EC00432=798156,1112951
EC00433=798156,1112951
EC00434=798156,1112951
EC00435=798156,1112951
EC00436=798156,1112951
EC00437=798156,1112951
EC00438=798156,1112951
EC00439=798156,1112951
EC00440=798156,1112951
EC00441=798156,1112951
EC00442=798156,1112951
EC00443=798156,1112951
EC00444=798156,1112951
EC00445=798156,1112951
EC00446=798156,1112951
EC00447=798156,1112951
EC00448=798156,1112951
EC00449=798156,1112951
EC00450=798156,1112951
EC00451=798156,1112951
EC00452=798156,1112951
EC00453=798156,1112951
EC00454=798156,1112951
EC00455=798156,1112951
EC00456=798156,1112951
EC00457=798156,1112951
EC00458=798156,1112951
EC00459=798156,1112951
EC00460=798156,1112951
EC00461=798156,1112951
EC00462=798156,1112951
EC00463=798156,1112951
EC00464=798156,1112951
EC00465=798156,1112951
EC00466=798156,1112951
EC00467=798156,1112951
EC00468=798156,1112951
EC00469=798156,1112951
EC00470=798156,1112951
EC00471=798156,1112951
EC00472=798155,1112950
EC00473=798155,1112950
EC00474=798156,1112951
EC00475=798156,1112951
EC00476=798156,1112951
EC00477=798156,1112951
EC00478=798156,1112951
EC00479=798156,1112951
EC00480=798155,1112951
EC00481=798155,1112951
EC00482=798156,1112951
EC00483=798156,1112951
EC00484=798156,1112951
EC00485=798156,1112951
EC00486=798156,1112951
EC00487=798156,1112951
EC00488=798156,1112951
EC00489=798156,1112951
EC00490=798155,1112950
EC00491=798156,1112951
EC00492=798156,1112951
EC00493=798156,1112951
EC00494=798156,1112951
EC00495=798156,1112951
EC00496=798156,1112951
EC00497=798156,1112951
EC00498=798156,1112951
EC00499=798156,1112951
EC00500=798156,1112951
EC00501=798156,1112951
EC00502=798156,1112951
EC00503=798156,1112951
EC00504=798156,1112951
EC00505=798156,1112951
EC00506=798156,1112951
EC00507=798155,1112950
EC00508=798156,1112951
EC00509=798156,1112951
EC00510=798156,1112951
EC00511=798156,1112951
EC00512=798156,1112951
EC00513=798156,1112951
EC00514=798156,1112951
EC00515=798156,1112951
EC00516=798156,1112951
EC00517=798156,1112951
EC00518=798155,1112950
EC00519=798156,1112951
EC00520=798156,1112951
EC00521=798156,1112951
EC00522=798156,1112951
EC00523=798156,1112951
EC00524=798156,1112951
EC00525=798156,1112951
EC00526=798156,1112951
EC00527=798156,1112951
EC00528=798156,1112951
EC00529=798156,1112951
EC00530=798156,1112951
EC00531=798156,1112951
EC00532=798156,1112951
EC00533=798156,1112951
EC00534=798156,1112951
EC00535=798156,1112951
EC00536=798156,1112951
EC00537=798156,1112951
EC00538=798156,1112951
EC00539=798156,1112951
EC00540=798156,1112951
EC00541=798156,1112951
EC00542=798156,1112951
EC00543=798156,1112951
EC00544=798156,1112951
EC00545=798156,1112951
EC00546=798156,1112951
EC00547=798156,1112951
EC00548=798156,1112951
EC00549=798156,1112951
EC00550=798156,1112951
EC00551=798155,1112950
EC00552=798156,1112951
EC00553=798156,1112951
EC00554=798154,1112949
EC00555=798156,1112951
EC00556=798156,1112951
EC00557=798156,1112951
EC00558=798156,1112951
EC00559=798156,1112951
EC00560=798156,1112951
EC00561=798156,1112951
EC00562=798156,1112951
EC00563=798156,1112951
EC00564=798156,1112951
EC00565=798156,1112951
EC00566=798156,1112951
EC00567=798156,1112951
EC00568=798156,1112951
EC00569=798156,1112951
EC00570=798156,1112951
EC00571=798156,1112951
EC00572=798156,1112951
EC00573=798156,1112951
EC00574=798156,1112951
EC00575=798156,1112951
EC00576=798156,1112951
EC00577=798156,1112951
EC00578=798156,1112951
EC00579=798156,1112951
EC00580=798156,1112951
EC00581=798156,1112951
EC00582=798156,1112951
EC00583=798156,1112951
EC00584=798156,1112951
EC00585=798156,1112951
EC00586=798156,1112951
EC00587=798156,1112951
EC00588=798156,1112951
EC00589=798156,1112951
EC00590=798156,1112951
EC00591=798156,1112951
EC00592=798156,1112951
EC00593=798156,1112951
EC00594=798156,1112951
EC00595=798156,1112951
EC00596=798156,1112951
EC00597=798156,1112951
EC00598=798156,1112951
EC00599=798156,1112951
EC00600=798156,1112951
EC00601=798156,1112951
EC00602=798156,1112951
EC00603=798156,1112951
EC00604=798156,1112951
EC00605=798156,1112951
EC00606=798156,1112951
EC00607=798156,1112951
EC00608=798156,1112951
EC00609=798156,1112951
EC00610=798156,1112951
EC00611=798156,1112951
EC00612=798156,1112951
EC00613=798156,1112951
EC00614=798156,1112951
EC00615=798156,1112951
EC00616=798156,1112951
EC00617=798156,1112951
EC00618=798156,1112951
EC00619=798155,1112951
EC00620=798156,1112951
EC00621=798156,1112951
EC00622=798156,1112951
EC00623=798156,1112951
EC00624=798156,1112951
EC00625=798156,1112951
EC00626=798156,1112951
EC00627=798156,1112951
EC00628=798156,1112951
EC00629=798156,1112951
EC00630=798156,1112951
EC00631=798156,1112951
EC00632=798156,1112951
EC00633=798156,1112951
EC00634=798156,1112951
EC00635=798156,1112951
EC00636=798156,1112951
EC00637=798156,1112951
EC00638=798156,1112951
EC00639=798156,1112951
EC00640=798156,1112951
EC00641=798156,1112951
EC00642=798156,1112951
EC00643=798156,1112951
EC00644=798156,1112951
EC00645=798156,1112951
EC00646=798156,1112951
EC00647=798156,1112951
EC00648=798156,1112951
EC00649=798156,1112951
EC00650=798156,1112951
EC00651=798156,1112951
EC00652=798156,1112951
EC00653=798156,1112951
EC00654=798156,1112951
EC00655=798156,1112951
EC00656=798156,1112951
EC00657=798156,1112951
EC00658=798156,1112951
EC00659=798156,1112951
EC00660=798156,1112951
EC00661=798156,1112951
EC00662=798156,1112951
EC00663=798156,1112951
EC00664=798156,1112951
EC00665=798156,1112951
EC00666=798156,1112951
EC00667=798156,1112951
EC00668=798156,1112951
EC00669=798156,1112951
EC00670=798156,1112951
EC00671=798156,1112951
EC00672=798156,1112951
EC00673=798156,1112951
EC00674=798156,1112951
EC00675=798156,1112951
EC00676=798156,1112951
EC00677=798156,1112951
EC00678=798156,1112951
EC00679=798156,1112951
EC00680=798156,1112951
EC00681=798156,1112951
EC00682=798156,1112951
EC00683=798156,1112951
EC00684=798156,1112951
EC00685=798156,1112951
EC00686=798156,1112951
EC00687=798156,1112951
EC00688=798156,1112951
EC00689=798156,1112951
EC00690=798156,1112951
EC00691=798156,1112951
EC00692=798156,1112951
EC00693=798156,1112951
EC00694=798156,1112951
EC00695=798156,1112951
EC00696=798156,1112951
EC00697=798156,1112951
EC00698=798156,1112951
EC00699=798156,1112951
EC00700=798156,1112951
EC00701=798156,1112951
EC00702=798156,1112951
EC00703=798156,1112951
EC00704=798156,1112951
EC00705=798156,1112951
EC00706=798156,1112951
EC00707=798155,1112950
EC00708=798155,1112950
EC00709=798155,1112950
EC00710=798156,1112951
EC00711=798156,1112951
EC00712=798156,1112951
EC00713=798156,1112951
EC00714=798156,1112951
EC00715=798156,1112951
EC00716=798156,1112951
EC00717=798156,1112951
EC00718=798156,1112951
EC00719=798156,1112951
EC00720=798156,1112951
EC00721=798156,1112951
EC00722=798156,1112951
EC00723=798156,1112951
EC00724=798156,1112951
EC00725=798156,1112951
EC00726=798156,1112951
EC00727=798156,1112951
EC00728=798156,1112951
EC00729=798156,1112951
EC00730=798156,1112951
EC00731=798156,1112951
EC00732=798156,1112951
EC00733=798156,1112951
EC00734=798156,1112951
EC00735=798156,1112951
EC00736=798156,1112951
EC00737=798156,1112951
EC00738=798156,1112951
EC00739=798156,1112951
EC00740=798156,1112951
EC00741=798156,1112951
EC00742=798156,1112951
EC00743=798156,1112951
EC00744=798156,1112951
EC00745=798156,1112951
EC00746=798156,1112951
EC00747=798156,1112951
EC00748=798156,1112951
EC00749=798156,1112951
EC00750=798156,1112951
EC00751=798156,1112951
EC00752=798156,1112951
EC00753=798156,1112951
EC00754=798155,1112950
EC00755=798156,1112951
EC00756=798156,1112951
EC00757=798156,1112951
EC00758=798156,1112951
EC00759=798156,1112951
EC00760=798156,1112951
EC00761=798156,1112951
EC00762=798156,1112951
EC00763=798156,1112951
EC00764=798156,1112951
EC00765=798156,1112951
EC00766=798156,1112951
EC00767=798156,1112951
EC00768=798156,1112951
EC00769=798156,1112951
EC00770=798156,1112951
EC00771=798156,1112951
EC00772=798156,1112951
EC00773=798156,1112951
EC00774=798156,1112951
EC00775=798156,1112951
EC00776=798156,1112951
EC00777=798156,1112951
EC00778=798156,1112951
EC00779=798156,1112951
EC00780=798156,1112951
EC00781=798156,1112951
EC00782=798156,1112951
EC00783=798156,1112951
EC00784=798156,1112951
EC00785=798156,1112951
EC00786=798156,1112951
EC00787=798156,1112951
EC00788=798156,1112951
EC00789=798156,1112951
EC00790=798156,1112951
EC00791=798156,1112951
EC00792=798156,1112951
EC00793=798156,1112951
EC00794=798156,1112951
EC00795=798156,1112951
EC00796=798156,1112951
EC00797=798156,1112951
EC00798=798156,1112951
EC00799=798156,1112951
EC00800=798156,1112951
EC00801=798156,1112951
EC00802=798156,1112951
EC00803=798156,1112951
EC00804=798156,1112951
EC00805=798156,1112951
EC00806=798156,1112951
EC00807=798156,1112951
EC00808=798156,1112951
EC00809=798156,1112951
EC00810=798156,1112951
EC00811=798156,1112951
EC00812=798156,1112951
EC00813=798156,1112951
EC00814=798156,1112951
EC00815=798156,1112951
EC00816=798156,1112951
EC00817=798156,1112951
EC00818=798156,1112951
EC00819=798156,1112951
EC00820=798156,1112951
EC00821=798156,1112951
EC00822=798156,1112951
EC00823=798156,1112951
EC00824=798156,1112951
EC00825=798156,1112951
EC00826=798156,1112951
EC00827=798156,1112951
EC00828=798156,1112951
EC00829=798156,1112951
EC00830=798156,1112951
EC00831=798156,1112951
EC00832=798156,1112951
EC00833=798156,1112951
EC00834=798156,1112951
EC00835=798156,1112951
EC00836=798156,1112951
EC00837=798156,1112951
EC00838=798156,1112951
EC00839=798156,1112951
EC00840=798156,1112951
EC00841=798156,1112951
EC00842=798156,1112951
EC00843=798156,1112951
EC00844=798156,1112951
EC00845=798156,1112951
EC00846=798156,1112951
EC00847=798156,1112951
EC00848=798156,1112951
EC00849=798156,1112951
EC00850=798156,1112951
EC00851=798156,1112951
EC00852=798156,1112951
EC00853=798156,1112951
EC00854=798156,1112951
EC00855=798156,1112951
EC00856=798156,1112951
EC00857=798156,1112951
EC00858=798156,1112951
EC00859=798156,1112951
EC00860=798156,1112951
EC00861=798156,1112951
EC00862=798156,1112951
EC00863=798156,1112951
EC00864=798156,1112951
EC00865=798156,1112951
EC00866=798156,1112951
EC00867=798156,1112951
EC00868=798156,1112951
EC00869=798155,1112951
EC00870=798155,1112951
EC00871=798156,1112951
EC00872=798156,1112951
EC00873=798156,1112951
EC00874=798156,1112951
EC00875=798156,1112951
EC00876=798156,1112951
EC00877=798156,1112951
EC00878=798156,1112951
EC00879=798155,1112950
EC00880=798155,1112950
EC00881=798155,1112950
EC00882=798155,1112950
EC00883=798155,1112950
EC00884=798156,1112951
EC00885=798156,1112951
EC00886=798156,1112951
EC00887=798156,1112951
EC00888=798156,1112951
EC00889=798156,1112951
EC00890=798156,1112951
EC00891=798156,1112951
EC00892=798156,1112951
EC00893=798156,1112951
EC00894=798156,1112951
EC00895=798156,1112951
EC00896=798156,1112951
EC00897=798156,1112951
EC00898=798156,1112951
EC00899=798156,1112951
EC00900=798156,1112951
EC00901=798156,1112951
EC00902=798156,1112951
EC00903=798156,1112951
EC00904=798156,1112951
EC00905=798156,1112951
EC00906=798156,1112951
EC00907=798156,1112951
EC00908=798156,1112951
EC00909=798156,1112951
EC00910=798156,1112951
EC00911=798156,1112951
EC00912=798156,1112951
EC00913=798156,1112951
EC00914=798156,1112951
EC00915=798156,1112951
EC00916=798156,1112951
EC00917=798156,1112951
EC00918=798156,1112951
EC00919=798156,1112951
EC00920=798156,1112951
EC00921=798156,1112951
EC00922=798156,1112951
EC00923=798156,1112951
EC00924=798156,1112951
EC00925=798156,1112951
EC00926=798156,1112951
EC00927=798156,1112951
EC00928=798156,1112951
EC00929=798156,1112951
EC00930=798156,1112951
EC00931=798156,1112951
EC00932=798156,1112951
EC00933=798156,1112951
EC00934=798156,1112951
EC00935=798156,1112951
EC00936=798156,1112951
EC00937=798156,1112951
EC00938=798156,1112951
EC00939=798156,1112951
EC00940=798156,1112951
EC00941=798156,1112951
EC00942=798156,1112951
EC00943=798156,1112951
EC00944=798156,1112951
EC00945=798156,1112951
EC00946=798156,1112951
EC00947=798156,1112951
EC00948=798156,1112951
EC00949=798156,1112951
EC00950=798156,1112951
EC00951=798156,1112951
EC00952=798156,1112951
EC00953=798156,1112951
EC00954=798156,1112951
EC00955=798156,1112951
EC00956=798156,1112951
EC00957=798156,1112951
EC00958=798156,1112951
EC00959=798156,1112951
EC00960=798156,1112951
EC00961=798156,1112951
EC00962=798156,1112951
EC00963=798156,1112951
EC00964=798156,1112951
EC00965=798156,1112951
EC00966=798156,1112951
EC00967=798156,1112951
EC00968=798156,1112951
EC00969=798156,1112951
EC00970=798156,1112951
EC00971=798156,1112951
EC00972=798156,1112951
EC00973=798156,1112951
EC00974=798156,1112951
EC00975=798156,1112951
EC00976=798156,1112951
EC00977=798156,1112951
EC00978=798156,1112951
EC00979=798156,1112951
EC00980=798156,1112951
EC00981=798156,1112951
EC00982=798156,1112951
EC00983=798156,1112951
EC00984=798156,1112951
EC00985=798156,1112951
EC00986=798156,1112951
EC00987=798156,1112951
EC00988=798156,1112951
EC00989=798156,1112951
EC00990=798156,1112951
EC00991=798156,1112951
EC00992=798156,1112951
EC00993=798156,1112951
EC00994=798156,1112951
EC00995=798156,1112951
EC00996=798156,1112949
EC00997=798156,1112951
EC00998=798156,1112951
EC00999=798156,1112951
EC01000=798156,1112951
EC01001=798156,1112951
EC01002=798156,1112951
EC01003=798156,1112951
EC01004=798156,1112951
EC01005=798156,1112951
EC01006=798156,1112951
EC01007=798156,1112951
EC01008=798156,1112951
EC01009=798156,1112951
EC01010=798156,1112951
EC01011=798156,1112951
EC01012=798156,1112951
EC01013=798156,1112951
EC01014=798156,1112951
EC01015=798156,1112951
EC01016=798156,1112951
EC01017=798156,1112951
EC01018=798156,1112951
EC01019=798156,1112951
EC01020=798156,1112951
EC01021=798156,1112951
EC01022=798156,1112951
EC01023=798156,1112951
EC01024=798156,1112951
EC01025=798156,1112951
EC01026=798156,1112951
EC01027=798156,1112951
EC01028=798156,1112951
EC01029=798156,1112951
EC01030=798156,1112951
EC01031=798156,1112951
EC01032=798156,1112951
EC01033=798156,1112951
EC01034=798156,1112951
EC01035=798156,1112951
EC01036=798156,1112951
EC01037=798156,1112951
EC01038=798156,1112951
EC01039=798156,1112951
EC01040=798156,1112951
EC01041=798156,1112951
EC01042=798156,1112951
EC01043=798156,1112951
EC01044=798156,1112951
EC01045=798156,1112951
EC01046=798156,1112951
EC01047=798156,1112951
EC01048=798156,1112951
EC01049=798156,1112951
EC01050=798156,1112951
EC01051=798156,1112951
EC01052=798156,1112951
EC01053=798156,1112951
EC01054=798156,1112951
EC01055=798156,1112951
EC01056=798156,1112951
EC01057=798156,1112951
EC01058=798156,1112951
EC01059=798156,1112951
EC01060=798156,1112951
EC01061=798155,1112950
EC01062=798155,1112950
EC01063=798155,1112950
EC01064=798155,1112950
EC01065=798155,1112950
EC01066=798155,1112950
EC01067=798155,1112950
EC01068=798156,1112951
EC01069=798156,1112951
EC01070=798156,1112951
EC01071=798156,1112951
EC01072=798156,1112951
EC01073=798156,1112951
EC01074=798156,1112951
EC01075=798156,1112951
EC01076=798156,1112951
EC01077=798156,1112951
EC01078=798156,1112951
EC01079=798156,1112951
EC01080=798156,1112951
EC01081=798156,1112951
EC01082=798156,1112951
EC01083=798156,1112951
EC01084=798156,1112951
EC01085=798156,1112951
EC01086=798156,1112951
EC01087=798156,1112951
EC01088=798156,1112951
EC01089=798156,1112951
EC01090=798156,1112951
EC01091=798156,1112951
EC01092=798156,1112951
EC01093=798156,1112951
EC01094=798156,1112951
EC01095=798156,1112951
EC01096=798156,1112951
EC01097=798156,1112951
EC01098=798156,1112951
EC01099=798156,1112951
EC01100=798156,1112951
EC01101=798156,1112951
EC01102=798156,1112951
EC01103=798156,1112951
EC01104=798156,1112951
EC01105=798156,1112951
EC01106=798156,1112951
EC01107=798156,1112951
EC01108=798156,1112951
EC01109=798156,1112951
EC01110=798156,1112951
EC01111=798156,1112951
EC01112=798156,1112951
EC01113=798156,1112951
EC01114=798156,1112951
EC01115=798156,1112951
EC01116=798156,1112951
EC01117=798156,1112951
EC01118=798156,1112951
EC01119=798156,1112951
EC01120=798156,1112951
EC01121=798156,1112951
EC01122=798156,1112951
EC01123=798156,1112951
EC01124=798156,1112951
EC01125=798156,1112951
EC01126=798156,1112951
EC01127=798156,1112951
EC01128=798156,1112951
EC01129=798156,1112951
EC01130=798156,1112951
EC01131=798156,1112951
EC01132=798156,1112951
EC01133=798156,1112951
EC01134=798156,1112951
EC01135=798155,1112949
EC01136=798156,1112951
EC01137=798156,1112951
EC01138=798156,1112951
EC01139=798156,1112951
EC01140=798156,1112951
EC01141=798156,1112951
EC01142=798156,1112951
EC01143=798156,1112951
EC01144=798156,1112951
EC01145=798156,1112951
EC01146=798156,1112951
EC01147=798156,1112951
EC01148=798156,1112951
EC01149=798156,1112951
EC01150=798156,1112951
EC01151=798156,1112951
EC01152=798156,1112951
EC01153=798156,1112951
///POSTYPE BASE
///RECTAN
///RCONF 0,0,0,0,0,0,0,0,0,0,0,0,0,0,0,0,0,0,0,0,0,0,0,0
P00006=0.222,-3.123,-1.508,0.0000,0.0000,0.0000
P00021=-0.225,-6.128,-0.405,0.0000,0.0000,0.0000
P00022=0.222,-3.123,-1.508,0.0000,0.0000,0.0000
P00023=0.143,-0.036,0.682,0.0000,0.0000,0.0000
P00024=0.145,-0.552,1.326,0.0000,0.0000,0.0000
P00025=-2.003,0.006,0.728,0.0000,0.0000,0.0000
P00026=0.562,-0.002,-0.337,0.0000,0.0000,0.0000
P00027=-0.746,0.015,-9.096,0.0000,0.0000,0.0000
P00028=-2.237,-0.018,-7.702,0.0000,0.0000,0.0000
P00029=-2.156,-0.086,-4.681,0.0000,0.0000,0.0000
P00030=5.926,-4.294,-1.390,0.0000,0.0000,0.0000
P00031=1.853,-0.001,-1.549,0.0000,0.0000,0.0000
P00032=1.957,0.503,-7.217,0.0000,0.0000,0.0000
///RCONF 0,0,0,0,1,0,0,0,0,0,0,0,0,0,0,0,0,0,0,0,0,0,0,0
P00033=-0.123,0.612,-5.012,0.0000,0.0000,0.0000
///RCONF 0,0,0,0,0,0,0,0,0,0,0,0,0,0,0,0,0,0,0,0,0,0,0,0
P00034=-0.304,0.773,-2.693,0.0000,0.0000,0.0000
P00035=2.817,0.591,-1.622,0.0000,0.0000,0.0000
P00036=-1.108,-0.829,1.850,0.0000,0.0000,0.0000
P00037=0.023,0.937,-2.677,0.0000,0.0000,0.0000
P00038=0.158,-1.133,-1.952,0.0000,0.0000,0.0000
P00039=0.012,-3.081,-0.106,0.0000,0.0000,0.0000
P00040=-0.030,9.648,2.467,0.0000,0.0000,0.0000
P00041=0.192,3.924,0.305,0.0000,0.0000,0.0000
P00042=-0.217,1.941,0.413,0.0000,0.0000,0.0000
P00043=-0.044,-1.937,1.197,0.0000,0.0000,0.0000
P00044=0.687,-2.322,1.156,0.0000,0.0000,0.0000
P00045=-0.068,-0.810,1.603,0.0000,0.0000,0.0000
P00046=0.799,0.043,1.292,0.0000,0.0000,0.0000
///RCONF 0,1,0,0,0,0,0,0,0,0,0,0,0,0,0,0,0,0,0,0,0,0,0,0
P00047=-0.011,1.737,-0.646,0.0000,0.0000,0.0000
///RCONF 0,0,0,0,0,0,0,0,0,0,0,0,0,0,0,0,0,0,0,0,0,0,0,0
P00048=2.411,0.025,-0.606,0.0000,0.0000,0.0000
P00049=3.413,-3.572,-1.618,0.0000,0.0000,0.0000
P00050=4.296,-4.501,-0.826,0.0000,0.0000,0.0000
P00051=0.367,3.892,0.009,0.0000,0.0000,0.0000
P00052=0.088,2.832,-0.342,0.0000,0.0000,0.0000
P00053=0.134,6.594,0.107,0.0000,0.0000,0.0000
P00054=-0.103,6.509,-0.702,0.0000,0.0000,0.0000
P00055=-0.342,8.912,1.324,0.0000,0.0000,0.0000
P00056=0.568,-0.032,0.830,0.0000,0.0000,0.0000
P00061=1.575,-3.405,-0.752,0.0000,0.0000,0.0000
P00062=-0.135,-0.848,-1.706,0.0000,0.0000,0.0000
P00063=0.036,-0.654,-3.005,0.0000,0.0000,0.0000
P00071=2.716,0.070,1.352,0.0000,0.0000,0.0000
P00072=1.041,-0.003,-0.797,0.0000,0.0000,0.0000
P00073=-0.961,5.319,-6.157,0.0000,0.0000,0.0000
P00074=1.123,1.944,-5.914,0.0000,0.0000,0.0000
P00080=-3.893,-3.240,-0.208,0.0000,0.0000,0.0000
P00081=19.486,11.347,1.262,0.0000,0.0000,0.0000
P00088=-2.376,0.094,2.453,0.0000,0.0000,0.0000
P00089=5.697,-3.100,-1.263,0.0000,0.0000,0.0000
P00095=-3.945,4.918,-0.177,0.0000,0.0000,0.0000
P00096=-0.633,5.398,-3.809,0.0000,0.0000,0.0000
P00097=0.069,0.776,0.128,0.0000,0.0000,0.0000
P00098=0.276,2.477,1.230,0.0000,0.0000,0.0000
P00105=-1.846,-0.871,-2.217,0.0000,0.0000,0.0000
//INST
///DATE 2025/04/07 05:36
///ATTR SC,RW
///GROUP1 RB1,BS1
///GROUP2 ST1
NOP
COMM CALL JOB:CLEAN-R1_KM_NEW
'X2_8B-21B(90,180)
'
MOVJ C00000 BC00000 VJ=100.00  +MOVJ EC00000 VJ=100.00
'Path S4722
SFTOF3D
MOVJ C00001 BC00001 VJ=100.00  +MOVJ EC00001 VJ=100.00
MOVL C00002 BC00002 V=666.7  +MOVJ EC00002 VJ=100.00
SMOVL C00003 BC00003 V=166.7  +MOVJ EC00003
SREFP 3 C00004 BC00004  +REFP EC00004
CALL JOB:SEARCH-R1-S13D
SET P095 P006
SFTON3D P095
SMOVL C00005 BC00005 V=166.7  +MOVJ EC00005
SREFP 3 C00006 BC00006  +REFP EC00006
CALL JOB:SEARCH-R1-S13D
SET P095 P006
SFTON3D P095
SMOVL C00007 BC00007 V=166.7  +MOVJ EC00007
MOVL C00008 BC00008 V=1000.0  +MOVJ EC00008 VJ=100.00
'EndPath S4722
'Path S4723
SFTOF3D
MOVJ C00009 BC00009 VJ=100.00  +MOVJ EC00009 VJ=100.00
MOVL C00010 BC00010 V=666.7  +MOVJ EC00010 VJ=100.00
SMOVL C00011 BC00011 V=166.7  +MOVJ EC00011
SREFP 3 C00012 BC00012  +REFP EC00012
CALL JOB:SEARCH-R1-S13D
SET P096 P006
SFTON3D P096
SMOVL C00013 BC00013 V=166.7  +MOVJ EC00013
SREFP 3 C00014 BC00014  +REFP EC00014
CALL JOB:SEARCH-R1-S13D
SET P096 P006
SFTON3D P096
SMOVL C00015 BC00015 V=166.7  +MOVJ EC00015
MOVL C00016 BC00016 V=1000.0  +MOVJ EC00016 VJ=100.00
'EndPath S4723
'
'
'Path S4093
SFTOF3D
MOVJ C00017 BC00017 VJ=100.00  +MOVJ EC00017 VJ=100.00
MOVL C00018 BC00018 V=666.7  +MOVJ EC00018 VJ=100.00
SMOVL C00019 BC00019 V=166.7  +MOVJ EC00019
SREFP 3 C00020 BC00020  +REFP EC00020
CALL JOB:SEARCH-R1-S13D
SET P097 P006
SFTON3D P097
SMOVL C00021 BC00021 V=166.7  +MOVJ EC00021
SREFP 3 C00022 BC00022  +REFP EC00022
CALL JOB:SEARCH-R1-S13D
SET P097 P006
SFTON3D P097
SMOVL C00023 BC00023 V=166.7  +MOVJ EC00023
SFTOF3D
MOVL C00024 BC00024 V=666.7  +MOVJ EC00024 VJ=100.00
SMOVL C00025 BC00025 V=166.7  +MOVJ EC00025
SREFP 3 C00026 BC00026  +REFP EC00026
CALL JOB:SEARCH-R1-S13D
SET P021 P006
SFTON3D P021
SMOVL C00027 BC00027 V=166.7  +MOVJ EC00027
SREFP 3 C00028 BC00028  +REFP EC00028
CALL JOB:SEARCH-R1-S13D
SET P021 P006
SFTON3D P021
SMOVL C00029 BC00029 V=166.7  +MOVJ EC00029
MOVL C00030 BC00030 V=1000.0  +MOVJ EC00030 VJ=100.00
'EndPath S4093
'Path S4094
SFTOF3D
MOVJ C00031 BC00031 VJ=100.00  +MOVJ EC00031 VJ=100.00
MOVL C00032 BC00032 V=666.7  +MOVJ EC00032 VJ=100.00
SMOVL C00033 BC00033 V=166.7  +MOVJ EC00033
SREFP 3 C00034 BC00034  +REFP EC00034
CALL JOB:SEARCH-R1-S13D
SET P022 P006
SFTON3D P022
SMOVL C00035 BC00035 V=166.7  +MOVJ EC00035
SREFP 3 C00036 BC00036  +REFP EC00036
CALL JOB:SEARCH-R1-S13D
SET P022 P006
SFTON3D P022
SMOVL C00037 BC00037 V=166.7  +MOVJ EC00037
MOVL C00038 BC00038 V=1000.0  +MOVJ EC00038 VJ=100.00
'EndPath S4094
MOVJ C00039 BC00039 VJ=100.00  +MOVJ EC00039 VJ=100.00
'Path S4205
SFTOF3D
MOVJ C00040 BC00040 VJ=100.00  +MOVJ EC00040 VJ=100.00
MOVL C00041 BC00041 V=666.7  +MOVJ EC00041 VJ=100.00
SMOVL C00042 BC00042 V=166.7  +MOVJ EC00042
SREFP 3 C00043 BC00043  +REFP EC00043
CALL JOB:SEARCH-R1-S13D
SET P050 P006
SFTON3D P050
SMOVL C00044 BC00044 V=166.7  +MOVJ EC00044
SREFP 3 C00045 BC00045  +REFP EC00045
CALL JOB:SEARCH-R1-S13D
SET P050 P006
SFTON3D P050
SMOVL C00046 BC00046 V=166.7  +MOVJ EC00046
SMOVL C00047 BC00047 V=250.0  +MOVJ EC00047
SMOVL C00048 BC00048 V=166.7  +MOVJ EC00048
SREFP 3 C00049 BC00049  +REFP EC00049
CALL JOB:SEARCH-R1-S13D
SET P050 P006
SFTON3D P050
SMOVL C00050 BC00050 V=250.0  +MOVJ EC00050
'EndPath S4205
'Path S4206
SFTOF3D
MOVL C00051 BC00051 V=1000.0  +MOVJ EC00051 VJ=100.00
SMOVL C00052 BC00052 V=166.7  +MOVJ EC00052
SREFP 3 C00053 BC00053  +REFP EC00053
CALL JOB:SEARCH-R1-S13D
SET P051 P006
SFTON3D P051
SMOVL C00054 BC00054 V=166.7  +MOVJ EC00054
SREFP 3 C00055 BC00055  +REFP EC00055
CALL JOB:SEARCH-R1-S13D
SET P051 P006
SFTON3D P051
SMOVL C00056 BC00056 V=166.7  +MOVJ EC00056
SMOVL C00057 BC00057 V=250.0  +MOVJ EC00057
SREFP 3 C00058 BC00058  +REFP EC00058
CALL JOB:SEARCH-R1-S13D
SET P051 P006
SFTON3D P051
SMOVL C00059 BC00059 V=250.0  +MOVJ EC00059
MOVL C00060 BC00060 V=1000.0  +MOVJ EC00060 VJ=100.00
'EndPath S4206
MOVJ C00061 BC00061 VJ=100.00  +MOVJ EC00061 VJ=100.00
'Path S4207
SFTOF3D
MOVJ C00062 BC00062 VJ=100.00  +MOVJ EC00062 VJ=100.00
MOVL C00063 BC00063 V=666.7  +MOVJ EC00063 VJ=100.00
SMOVL C00064 BC00064 V=166.7  +MOVJ EC00064
SREFP 3 C00065 BC00065  +REFP EC00065
CALL JOB:SEARCH-R1-S13D
SET P054 P006
SFTON3D P054
SMOVL C00066 BC00066 V=250.0  +MOVJ EC00066
SMOVL C00067 BC00067 V=233.3  +MOVJ EC00067
SMOVL C00068 BC00068 V=166.7  +MOVJ EC00068
SREFP 3 C00069 BC00069  +REFP EC00069
CALL JOB:SEARCH-R1-S13D
SET P054 P006
SFTON3D P054
SMOVL C00070 BC00070 V=166.7  +MOVJ EC00070
SMOVL C00071 BC00071 V=416.7  +MOVJ EC00071
SMOVL C00072 BC00072 V=250.0  +MOVJ EC00072
SREFP 3 C00073 BC00073  +REFP EC00073
CALL JOB:SEARCH-R1-S13D
SET P054 P006
SFTON3D P054
SMOVL C00074 BC00074 V=250.0  +MOVJ EC00074
MOVL C00075 BC00075 V=1000.0  +MOVJ EC00075 VJ=100.00
'EndPath S4207
'Path S4095
SFTOF3D
MOVJ C00076 BC00076 VJ=100.00  +MOVJ EC00076 VJ=100.00
MOVJ C00077 BC00077 VJ=100.00  +MOVJ EC00077 VJ=100.00
SMOVL C00078 BC00078 V=200.0  +MOVJ EC00078
SREFP 3 C00079 BC00079  +REFP EC00079
CALL JOB:SEARCH-R1-S13D
SET P089 P006
SFTON3D P089
SMOVL C00080 BC00080 V=166.7  +MOVJ EC00080
SMOVL C00081 BC00081 V=166.7  +MOVJ EC00081
SREFP 3 C00082 BC00082  +REFP EC00082
CALL JOB:SEARCH-R1-S13D
SET P089 P006
SFTON3D P089
SMOVL C00083 BC00083 V=166.7  +MOVJ EC00083
SMOVL C00084 BC00084 V=166.7  +MOVJ EC00084
SREFP 3 C00085 BC00085  +REFP EC00085
CALL JOB:SEARCH-R1-S13D
SET P089 P006
SFTON3D P089
SMOVL C00086 BC00086 V=166.7  +MOVJ EC00086
SMOVL C00087 BC00087 V=1000.0  +MOVJ EC00087
SFTOF3D
MOVJ C00088 BC00088 VJ=100.00  +MOVJ EC00088 VJ=100.00
MOVL C00089 BC00089 V=666.7  +MOVJ EC00089 VJ=100.00
SMOVL C00090 BC00090 V=166.7  +MOVJ EC00090
SREFP 3 C00091 BC00091  +REFP EC00091
CALL JOB:SEARCH-R1-S13D
SET P034 P006
SFTON3D P034
SMOVL C00092 BC00092 V=250.0  +MOVJ EC00092
SMOVL C00093 BC00093 V=233.3  +MOVJ EC00093
SMOVL C00094 BC00094 V=166.7  +MOVJ EC00094
SREFP 3 C00095 BC00095  +REFP EC00095
CALL JOB:SEARCH-R1-S13D
SET P034 P006
SFTON3D P034
SMOVL C00096 BC00096 V=166.7  +MOVJ EC00096
SMOVL C00097 BC00097 V=166.7  +MOVJ EC00097
SREFP 3 C00098 BC00098  +REFP EC00098
CALL JOB:SEARCH-R1-S13D
SET P034 P006
SFTON3D P034
SMOVL C00099 BC00099 V=166.7  +MOVJ EC00099
MOVJ C00100 BC00100 VJ=50.00  +MOVJ EC00100 VJ=30.00
'EndPath S4095
'Path S4096
SFTOF3D
MOVJ C00101 BC00101 VJ=50.00  +MOVJ EC00101 VJ=30.00
MOVJ C00102 BC00102 VJ=50.00  +MOVJ EC00102 VJ=30.00
MOVJ C00103 BC00103 VJ=50.00  +MOVJ EC00103 VJ=30.00
SMOVL C00104 BC00104 V=166.7  +MOVJ EC00104
SREFP 3 C00105 BC00105  +REFP EC00105
CALL JOB:SEARCH-R1-S13D
SET P061 P006
SFTON3D P061
SMOVL C00106 BC00106 V=166.7  +MOVJ EC00106
SREFP 3 C00107 BC00107  +REFP EC00107
CALL JOB:SEARCH-R1-S13D
SET P061 P006
SFTON3D P061
SMOVL C00108 BC00108 V=166.7  +MOVJ EC00108
SFTOF3D
SMOVL C00109 BC00109 V=666.7  +MOVJ EC00109
SMOVL C00110 BC00110 V=166.7  +MOVJ EC00110
SREFP 3 C00111 BC00111  +REFP EC00111
CALL JOB:SEARCH-R1-S13D
SET P062 P006
SFTON3D P062
SMOVL C00112 BC00112 V=166.7  +MOVJ EC00112
SREFP 3 C00113 BC00113  +REFP EC00113
CALL JOB:SEARCH-R1-S13D
SET P062 P006
SFTON3D P062
SMOVL C00114 BC00114 V=250.0  +MOVJ EC00114
SFTOF3D
SMOVL C00115 BC00115 V=500.0  +MOVJ EC00115
SMOVL C00116 BC00116 V=166.7  +MOVJ EC00116
SREFP 3 C00117 BC00117  +REFP EC00117
CALL JOB:SEARCH-R1-S13D
SET P063 P006
SFTON3D P063
SMOVL C00118 BC00118 V=166.7  +MOVJ EC00118
SREFP 3 C00119 BC00119  +REFP EC00119
CALL JOB:SEARCH-R1-S13D
SET P063 P006
SFTON3D P063
SMOVL C00120 BC00120 V=166.7  +MOVJ EC00120
SFTOF3D
SMOVL C00121 BC00121 V=1000.0  +MOVJ EC00121
MOVJ C00122 BC00122 VJ=100.00  +MOVJ EC00122 VJ=30.00
MOVJ C00123 BC00123 VJ=50.00  +MOVJ EC00123 VJ=30.00
MOVJ C00124 BC00124 VJ=100.00  +MOVJ EC00124 VJ=100.00
MOVL C00125 BC00125 V=666.7  +MOVJ EC00125 VJ=100.00
SMOVL C00126 BC00126 V=166.7  +MOVJ EC00126
SREFP 3 C00127 BC00127  +REFP EC00127
CALL JOB:SEARCH-R1-S13D
SET P023 P006
SFTON3D P023
SMOVL C00128 BC00128 V=166.7  +MOVJ EC00128
SMOVL C00129 BC00129 V=333.3  +MOVJ EC00129
SMOVL C00130 BC00130 V=166.7  +MOVJ EC00130
SREFP 3 C00131 BC00131  +REFP EC00131
CALL JOB:SEARCH-R1-S13D
SET P023 P006
SFTON3D P023
SMOVL C00132 BC00132 V=166.7  +MOVJ EC00132
SMOVL C00133 BC00133 V=166.7  +MOVJ EC00133
SREFP 3 C00134 BC00134  +REFP EC00134
CALL JOB:SEARCH-R1-S13D
SET P023 P006
SFTON3D P023
SMOVL C00135 BC00135 V=166.7  +MOVJ EC00135
MOVL C00136 BC00136 V=1000.0  +MOVJ EC00136 VJ=100.00
'EndPath S4096
MOVJ C00137 BC00137 VJ=100.00  +MOVJ EC00137 VJ=100.00
'Path S4097
SFTOF3D
MOVJ C00138 BC00138 VJ=100.00  +MOVJ EC00138 VJ=100.00
MOVL C00139 BC00139 V=666.7  +MOVJ EC00139 VJ=100.00
SMOVL C00140 BC00140 V=166.7  +MOVJ EC00140
SREFP 3 C00141 BC00141  +REFP EC00141
CALL JOB:SEARCH-R1-S13D
SET P024 P006
SFTON3D P024
SMOVL C00142 BC00142 V=166.7  +MOVJ EC00142
SREFP 3 C00143 BC00143  +REFP EC00143
CALL JOB:SEARCH-R1-S13D
SET P024 P006
SFTON3D P024
SMOVL C00144 BC00144 V=166.7  +MOVJ EC00144
SMOVL C00145 BC00145 V=166.7  +MOVJ EC00145
SREFP 3 C00146 BC00146  +REFP EC00146
CALL JOB:SEARCH-R1-S13D
SET P024 P006
SFTON3D P024
SMOVL C00147 BC00147 V=166.7  +MOVJ EC00147
SMOVL C00148 BC00148 V=166.7  +MOVJ EC00148
MOVL C00149 BC00149 V=666.7  +MOVJ EC00149 VJ=100.00
SMOVL C00150 BC00150 V=166.7  +MOVJ EC00150
SREFP 3 C00151 BC00151  +REFP EC00151
CALL JOB:SEARCH-R1-S13D
SET P105 P006
SFTON3D P105
SMOVL C00152 BC00152 V=166.7  +MOVJ EC00152
SREFP 3 C00153 BC00153  +REFP EC00153
CALL JOB:SEARCH-R1-S13D
SET P105 P006
SFTON3D P105
SMOVL C00154 BC00154 V=166.7  +MOVJ EC00154
MOVL C00155 BC00155 V=1000.0  +MOVJ EC00155 VJ=100.00
'EndPath S4097
'Path S4098
SFTOF3D
SMOVL C00156 BC00156 V=666.7  +MOVJ EC00156
SMOVL C00157 BC00157 V=166.7  +MOVJ EC00157
SREFP 3 C00158 BC00158  +REFP EC00158
CALL JOB:SEARCH-R1-S13D
SET P036 P006
SFTON3D P036
SMOVL C00159 BC00159 V=166.7  +MOVJ EC00159
SREFP 3 C00160 BC00160  +REFP EC00160
CALL JOB:SEARCH-R1-S13D
SET P036 P006
SFTON3D P036
SMOVL C00161 BC00161 V=166.7  +MOVJ EC00161
SFTOF3D
MOVJ C00162 BC00162 VJ=100.00  +MOVJ EC00162 VJ=100.00
MOVL C00163 BC00163 V=666.7  +MOVJ EC00163 VJ=100.00
SMOVL C00164 BC00164 V=166.7  +MOVJ EC00164
SREFP 3 C00165 BC00165  +REFP EC00165
CALL JOB:SEARCH-R1-S13D
SET P035 P006
SFTON3D P035
SMOVL C00166 BC00166 V=166.7  +MOVJ EC00166
SREFP 3 C00167 BC00167  +REFP EC00167
CALL JOB:SEARCH-R1-S13D
SET P035 P006
SFTON3D P035
SMOVL C00168 BC00168 V=166.7  +MOVJ EC00168
SMOVL C00169 BC00169 V=166.7  +MOVJ EC00169
SMOVL C00170 BC00170 V=166.7  +MOVJ EC00170
SREFP 3 C00171 BC00171  +REFP EC00171
CALL JOB:SEARCH-R1-S13D
SET P035 P006
SFTON3D P035
SMOVL C00172 BC00172 V=166.7  +MOVJ EC00172
MOVL C00173 BC00173 V=1000.0  +MOVJ EC00173 VJ=100.00
'EndPath S4098
'Path S4099
SFTOF3D
MOVJ C00174 BC00174 VJ=100.00  +MOVJ EC00174 VJ=100.00
MOVL C00175 BC00175 V=666.7  +MOVJ EC00175 VJ=100.00
SMOVL C00176 BC00176 V=166.7  +MOVJ EC00176
SREFP 3 C00177 BC00177  +REFP EC00177
CALL JOB:SEARCH-R1-S13D
SET P029 P006
SFTON3D P029
SMOVL C00178 BC00178 V=166.7  +MOVJ EC00178
SREFP 3 C00179 BC00179  +REFP EC00179
CALL JOB:SEARCH-R1-S13D
SET P029 P006
SFTON3D P029
SMOVL C00180 BC00180 V=166.7  +MOVJ EC00180
SMOVL C00181 BC00181 V=250.0  +MOVJ EC00181
SMOVL C00182 BC00182 V=166.7  +MOVJ EC00182
SREFP 3 C00183 BC00183  +REFP EC00183
CALL JOB:SEARCH-R1-S13D
SET P037 P006
SFTON3D P037
SMOVL C00184 BC00184 V=166.7  +MOVJ EC00184
SREFP 3 C00185 BC00185  +REFP EC00185
CALL JOB:SEARCH-R1-S13D
SET P037 P006
SFTON3D P037
SMOVL C00186 BC00186 V=166.7  +MOVJ EC00186
SMOVL C00187 BC00187 V=166.7  +MOVJ EC00187
SREFP 3 C00188 BC00188  +REFP EC00188
CALL JOB:SEARCH-R1-S13D
SET P038 P006
SFTON3D P038
SMOVL C00189 BC00189 V=166.7  +MOVJ EC00189
SREFP 3 C00190 BC00190  +REFP EC00190
CALL JOB:SEARCH-R1-S13D
SET P038 P006
SFTON3D P038
SMOVL C00191 BC00191 V=166.7  +MOVJ EC00191
'EndPath S4099
'Path S4855
SFTOF3D
MOVL C00192 BC00192 V=666.7  +MOVJ EC00192 VJ=100.00
SMOVL C00193 BC00193 V=166.7  +MOVJ EC00193
SREFP 3 C00194 BC00194  +REFP EC00194
CALL JOB:SEARCH-R1-S13D
SET P039 P006
SFTON3D P039
SMOVL C00195 BC00195 V=166.7  +MOVJ EC00195
SREFP 3 C00196 BC00196  +REFP EC00196
CALL JOB:SEARCH-R1-S13D
SET P039 P006
SFTON3D P039
SMOVL C00197 BC00197 V=166.7  +MOVJ EC00197
SMOVL C00198 BC00198 V=250.0  +MOVJ EC00198
SMOVL C00199 BC00199 V=166.7  +MOVJ EC00199
SREFP 3 C00200 BC00200  +REFP EC00200
CALL JOB:SEARCH-R1-S13D
SET P040 P006
SFTON3D P040
SMOVL C00201 BC00201 V=166.7  +MOVJ EC00201
SREFP 3 C00202 BC00202  +REFP EC00202
CALL JOB:SEARCH-R1-S13D
SET P040 P006
SFTON3D P040
SMOVL C00203 BC00203 V=166.7  +MOVJ EC00203
SMOVL C00204 BC00204 V=166.7  +MOVJ EC00204
SREFP 3 C00205 BC00205  +REFP EC00205
CALL JOB:SEARCH-R1-S13D
SET P041 P006
SFTON3D P041
SMOVL C00206 BC00206 V=166.7  +MOVJ EC00206
SREFP 3 C00207 BC00207  +REFP EC00207
CALL JOB:SEARCH-R1-S13D
SET P041 P006
SFTON3D P041
SMOVL C00208 BC00208 V=166.7  +MOVJ EC00208
'EndPath S4099
'Path S4855
SFTOF3D
MOVL C00209 BC00209 V=666.7  +MOVJ EC00209 VJ=100.00
SMOVL C00210 BC00210 V=166.7  +MOVJ EC00210
SREFP 3 C00211 BC00211  +REFP EC00211
CALL JOB:SEARCH-R1-S13D
SET P071 P006
SFTON3D P071
SMOVL C00212 BC00212 V=166.7  +MOVJ EC00212
SREFP 3 C00213 BC00213  +REFP EC00213
CALL JOB:SEARCH-R1-S13D
SET P071 P006
SFTON3D P071
SMOVL C00214 BC00214 V=166.7  +MOVJ EC00214
SMOVL C00215 BC00215 V=166.7  +MOVJ EC00215
SREFP 3 C00216 BC00216  +REFP EC00216
CALL JOB:SEARCH-R1-S13D
SET P071 P006
SFTON3D P071
SMOVL C00217 BC00217 V=166.7  +MOVJ EC00217
MOVL C00218 BC00218 V=1000.0  +MOVJ EC00218 VJ=100.00
MOVL C00219 BC00219 V=666.7  +MOVJ EC00219 VJ=100.00
SMOVL C00220 BC00220 V=166.7  +MOVJ EC00220
SREFP 3 C00221 BC00221  +REFP EC00221
CALL JOB:SEARCH-R1-S13D
SET P080 P006
SFTON3D P080
SMOVL C00222 BC00222 V=166.7  +MOVJ EC00222
SREFP 3 C00223 BC00223  +REFP EC00223
CALL JOB:SEARCH-R1-S13D
SET P080 P006
SFTON3D P080
SMOVL C00224 BC00224 V=166.7  +MOVJ EC00224
SMOVL C00225 BC00225 V=250.0  +MOVJ EC00225
SMOVL C00226 BC00226 V=166.7  +MOVJ EC00226
SREFP 3 C00227 BC00227  +REFP EC00227
CALL JOB:SEARCH-R1-S13D
SET P042 P006
SFTON3D P042
SMOVL C00228 BC00228 V=166.7  +MOVJ EC00228
SREFP 3 C00229 BC00229  +REFP EC00229
CALL JOB:SEARCH-R1-S13D
SET P042 P006
SFTON3D P042
SMOVL C00230 BC00230 V=166.7  +MOVJ EC00230
SMOVL C00231 BC00231 V=166.7  +MOVJ EC00231
SREFP 3 C00232 BC00232  +REFP EC00232
CALL JOB:SEARCH-R1-S13D
SET P043 P006
SFTON3D P043
SMOVL C00233 BC00233 V=166.7  +MOVJ EC00233
SREFP 3 C00234 BC00234  +REFP EC00234
CALL JOB:SEARCH-R1-S13D
SET P043 P006
SFTON3D P043
SMOVL C00235 BC00235 V=166.7  +MOVJ EC00235
'EndPath S4099
'Path S4855
SFTOF3D
MOVL C00236 BC00236 V=666.7  +MOVJ EC00236 VJ=100.00
SMOVL C00237 BC00237 V=166.7  +MOVJ EC00237
SREFP 3 C00238 BC00238  +REFP EC00238
CALL JOB:SEARCH-R1-S13D
SET P044 P006
SFTON3D P044
SMOVL C00239 BC00239 V=166.7  +MOVJ EC00239
SREFP 3 C00240 BC00240  +REFP EC00240
CALL JOB:SEARCH-R1-S13D
SET P044 P006
SFTON3D P044
SMOVL C00241 BC00241 V=166.7  +MOVJ EC00241
SMOVL C00242 BC00242 V=250.0  +MOVJ EC00242
SMOVL C00243 BC00243 V=166.7  +MOVJ EC00243
SREFP 3 C00244 BC00244  +REFP EC00244
CALL JOB:SEARCH-R1-S13D
SET P045 P006
SFTON3D P045
SMOVL C00245 BC00245 V=166.7  +MOVJ EC00245
SREFP 3 C00246 BC00246  +REFP EC00246
CALL JOB:SEARCH-R1-S13D
SET P045 P006
SFTON3D P045
SMOVL C00247 BC00247 V=166.7  +MOVJ EC00247
SMOVL C00248 BC00248 V=166.7  +MOVJ EC00248
SREFP 3 C00249 BC00249  +REFP EC00249
CALL JOB:SEARCH-R1-S13D
SET P046 P006
SFTON3D P046
SMOVL C00250 BC00250 V=166.7  +MOVJ EC00250
SREFP 3 C00251 BC00251  +REFP EC00251
CALL JOB:SEARCH-R1-S13D
SET P046 P006
SFTON3D P046
SMOVL C00252 BC00252 V=166.7  +MOVJ EC00252
'EndPath S4099
'Path S4855
SFTOF3D
PAUSE
MOVJ C00253 BC00253 VJ=100.00  +MOVJ EC00253 VJ=100.00
MOVL C00254 BC00254 V=666.7  +MOVJ EC00254 VJ=100.00
SMOVL C00255 BC00255 V=166.7  +MOVJ EC00255
SREFP 3 C00256 BC00256  +REFP EC00256
CALL JOB:SEARCH-R1-S13D
SET P072 P006
SFTON3D P072
SMOVL C00257 BC00257 V=166.7  +MOVJ EC00257
SREFP 3 C00258 BC00258  +REFP EC00258
CALL JOB:SEARCH-R1-S13D
SET P072 P006
SFTON3D P072
SMOVL C00259 BC00259 V=166.7  +MOVJ EC00259
MOVL C00260 BC00260 V=1000.0  +MOVJ EC00260 VJ=100.00
'EndPath S4856
MOVJ C00261 BC00261 VJ=100.00  +MOVJ EC00261 VJ=100.00
'Path S4857
SFTOF3D
MOVJ C00262 BC00262 VJ=100.00  +MOVJ EC00262 VJ=100.00
MOVJ C00263 BC00263 VJ=100.00  +MOVJ EC00263 VJ=100.00
MOVL C00264 BC00264 V=666.7  +MOVJ EC00264 VJ=100.00
SMOVL C00265 BC00265 V=166.7  +MOVJ EC00265
SREFP 3 C00266 BC00266  +REFP EC00266
CALL JOB:SEARCH-R1-S13D
SET P073 P006
SFTON3D P073
SMOVL C00267 BC00267 V=166.7  +MOVJ EC00267
SMOVL C00268 BC00268 V=166.7  +MOVJ EC00268
SREFP 3 C00269 BC00269  +REFP EC00269
CALL JOB:SEARCH-R1-S13D
SET P073 P006
SFTON3D P073
SMOVL C00270 BC00270 V=166.7  +MOVJ EC00270
SMOVL C00271 BC00271 V=166.7  +MOVJ EC00271
SREFP 3 C00272 BC00272  +REFP EC00272
CALL JOB:SEARCH-R1-S13D
SET P073 P006
SFTON3D P073
SMOVL C00273 BC00273 V=166.7  +MOVJ EC00273
MOVL C00274 BC00274 V=1000.0  +MOVJ EC00274 VJ=100.00
'EndPath S4857
MOVJ C00275 BC00275 VJ=100.00  +MOVJ EC00275 VJ=100.00
MOVJ C00276 BC00276 VJ=100.00  +MOVJ EC00276 VJ=100.00
'Path S4858
SFTOF3D
MOVJ C00277 BC00277 VJ=100.00  +MOVJ EC00277 VJ=100.00
MOVL C00278 BC00278 V=666.7  +MOVJ EC00278 VJ=100.00
SMOVL C00279 BC00279 V=166.7  +MOVJ EC00279
SREFP 3 C00280 BC00280  +REFP EC00280
CALL JOB:SEARCH-R1-S13D
SET P074 P006
SFTON3D P074
SMOVL C00281 BC00281 V=166.7  +MOVJ EC00281
SREFP 3 C00282 BC00282  +REFP EC00282
CALL JOB:SEARCH-R1-S13D
SET P074 P006
SFTON3D P074
SMOVL C00283 BC00283 V=166.7  +MOVJ EC00283
MOVL C00284 BC00284 V=1000.0  +MOVJ EC00284 VJ=100.00
'EndPath S4858
MOVJ C00285 BC00285 VJ=100.00  +MOVJ EC00285 VJ=100.00
MOVJ C00286 BC00286 VJ=100.00  +MOVJ EC00286 VJ=100.00
'Path S4100
SFTOF3D
MOVJ C00287 BC00287 VJ=100.00  +MOVJ EC00287 VJ=100.00
MOVL C00288 BC00288 V=666.7  +MOVJ EC00288 VJ=100.00
SMOVL C00289 BC00289 V=166.7  +MOVJ EC00289
SREFP 3 C00290 BC00290  +REFP EC00290
CALL JOB:SEARCH-R1-S13D
SET P081 P006
SFTON3D P081
SMOVL C00291 BC00291 V=166.7  +MOVJ EC00291
SREFP 3 C00292 BC00292  +REFP EC00292
CALL JOB:SEARCH-R1-S13D
SET P081 P006
SFTON3D P081
SMOVL C00293 BC00293 V=166.7  +MOVJ EC00293
SMOVL C00294 BC00294 V=666.7  +MOVJ EC00294
SMOVL C00295 BC00295 V=666.7  +MOVJ EC00295
SMOVL C00296 BC00296 V=666.7  +MOVJ EC00296
SMOVL C00297 BC00297 V=166.7  +MOVJ EC00297
SREFP 3 C00298 BC00298  +REFP EC00298
CALL JOB:SEARCH-R1-S13D
SET P081 P006
SFTON3D P081
SMOVL C00299 BC00299 V=250.0  +MOVJ EC00299
SMOVL C00300 BC00300 V=166.7  +MOVJ EC00300
SREFP 3 C00301 BC00301  +REFP EC00301
CALL JOB:SEARCH-R1-S13D
SET P047 P006
SFTON3D P047
SMOVL C00302 BC00302 V=250.0  +MOVJ EC00302
SREFP 3 C00303 BC00303  +REFP EC00303
CALL JOB:SEARCH-R1-S13D
SET P047 P006
SFTON3D P047
SMOVL C00304 BC00304 V=250.0  +MOVJ EC00304
SMOVL C00305 BC00305 V=250.0  +MOVJ EC00305
SREFP 3 C00306 BC00306  +REFP EC00306
CALL JOB:SEARCH-R1-S13D
SET P047 P006
SFTON3D P047
SMOVL C00307 BC00307 V=250.0  +MOVJ EC00307
SMOVL C00308 BC00308 V=166.7  +MOVJ EC00308
SREFP 3 C00309 BC00309  +REFP EC00309
CALL JOB:SEARCH-R1-S13D
SET P048 P006
SFTON3D P048
SMOVL C00310 BC00310 V=250.0  +MOVJ EC00310
SREFP 3 C00311 BC00311  +REFP EC00311
CALL JOB:SEARCH-R1-S13D
SET P048 P006
SFTON3D P048
SMOVL C00312 BC00312 V=250.0  +MOVJ EC00312
SMOVL C00313 BC00313 V=250.0  +MOVJ EC00313
SREFP 3 C00314 BC00314  +REFP EC00314
CALL JOB:SEARCH-R1-S13D
SET P048 P006
SFTON3D P048
SMOVL C00315 BC00315 V=250.0  +MOVJ EC00315
SMOVL C00316 BC00316 V=666.7  +MOVJ EC00316
SFTOF3D
SMOVL C00317 BC00317 V=666.7  +MOVJ EC00317
MOVJ C00318 BC00318 VJ=100.00  +MOVJ EC00318 VJ=100.00
MOVL C00319 BC00319 V=666.7  +MOVJ EC00319 VJ=100.00
SMOVL C00320 BC00320 V=166.7  +MOVJ EC00320
SREFP 3 C00321 BC00321  +REFP EC00321
CALL JOB:SEARCH-R1-S13D
SET P026 P006
SFTON3D P026
SMOVL C00322 BC00322 V=166.7  +MOVJ EC00322
SREFP 3 C00323 BC00323  +REFP EC00323
CALL JOB:SEARCH-R1-S13D
SET P026 P006
SFTON3D P026
SMOVL C00324 BC00324 V=166.7  +MOVJ EC00324
SMOVL C00325 BC00325 V=666.7  +MOVJ EC00325
SMOVL C00326 BC00326 V=666.7  +MOVJ EC00326
SMOVL C00327 BC00327 V=666.7  +MOVJ EC00327
SMOVL C00328 BC00328 V=166.7  +MOVJ EC00328
SREFP 3 C00329 BC00329  +REFP EC00329
CALL JOB:SEARCH-R1-S13D
SET P026 P006
SFTON3D P026
SMOVL C00330 BC00330 V=250.0  +MOVJ EC00330
SMOVL C00331 BC00331 V=666.7  +MOVJ EC00331
MOVL C00332 BC00332 V=1000.0  +MOVJ EC00332 VJ=100.00
'EndPath S4100
MOVJ C00333 BC00333 VJ=50.00  +MOVJ EC00333 VJ=100.00
'Path S4101
SFTOF3D
MOVJ C00334 BC00334 VJ=50.00  +MOVJ EC00334 VJ=100.00
MOVL C00335 BC00335 V=666.7  +MOVJ EC00335 VJ=100.00
SMOVL C00336 BC00336 V=166.7  +MOVJ EC00336
SREFP 3 C00337 BC00337  +REFP EC00337
CALL JOB:SEARCH-R1-S13D
SET P025 P006
SFTON3D P025
SMOVL C00338 BC00338 V=166.7  +MOVJ EC00338
SREFP 3 C00339 BC00339  +REFP EC00339
CALL JOB:SEARCH-R1-S13D
SET P025 P006
SFTON3D P025
SMOVL C00340 BC00340 V=166.7  +MOVJ EC00340
SMOVL C00341 BC00341 V=333.3  +MOVJ EC00341
SMOVL C00342 BC00342 V=166.7  +MOVJ EC00342
SREFP 3 C00343 BC00343  +REFP EC00343
CALL JOB:SEARCH-R1-S13D
SET P025 P006
SFTON3D P025
SMOVL C00344 BC00344 V=166.7  +MOVJ EC00344
MOVL C00345 BC00345 V=1000.0  +MOVJ EC00345 VJ=100.00
MOVL C00346 BC00346 V=666.7  +MOVJ EC00346 VJ=0.78
MOVL C00347 BC00347 V=666.7  +MOVJ EC00347 VJ=0.78
MOVL C00348 BC00348 V=666.7  +MOVJ EC00348 VJ=0.78
SMOVL C00349 BC00349 V=166.7  +MOVJ EC00349
SREFP 3 C00350 BC00350  +REFP EC00350
CALL JOB:SEARCH-R1-S13D
SET P049 P006
SFTON3D P049
SMOVL C00351 BC00351 V=166.7  +MOVJ EC00351
SREFP 3 C00352 BC00352  +REFP EC00352
CALL JOB:SEARCH-R1-S13D
SET P049 P006
SFTON3D P049
SMOVL C00353 BC00353 V=166.7  +MOVJ EC00353
MOVL C00354 BC00354 V=666.7  +MOVJ EC00354 VJ=0.78
SMOVL C00355 BC00355 V=166.7  +MOVJ EC00355
SREFP 3 C00356 BC00356  +REFP EC00356
CALL JOB:SEARCH-R1-S13D
SET P055 P006
SFTON3D P055
SMOVL C00357 BC00357 V=166.7  +MOVJ EC00357
SREFP 3 C00358 BC00358  +REFP EC00358
CALL JOB:SEARCH-R1-S13D
SET P055 P006
SFTON3D P055
SMOVL C00359 BC00359 V=166.7  +MOVJ EC00359
SFTOF3D
'EndPath S4101
MOVJ C00360 BC00360 VJ=100.00  +MOVJ EC00360 VJ=100.00
'Path S4102
SFTOF3D
MOVJ C00361 BC00361 VJ=100.00  +MOVJ EC00361 VJ=100.00
MOVL C00362 BC00362 V=666.7  +MOVJ EC00362 VJ=100.00
SMOVL C00363 BC00363 V=166.7  +MOVJ EC00363
SREFP 3 C00364 BC00364  +REFP EC00364
CALL JOB:SEARCH-R1-S13D
SET P028 P006
SFTON3D P028
SMOVL C00365 BC00365 V=166.7  +MOVJ EC00365
SREFP 3 C00366 BC00366  +REFP EC00366
CALL JOB:SEARCH-R1-S13D
SET P028 P006
SFTON3D P028
SMOVL C00367 BC00367 V=166.7  +MOVJ EC00367
SMOVL C00368 BC00368 V=333.3  +MOVJ EC00368
SMOVL C00369 BC00369 V=166.7  +MOVJ EC00369
SREFP 3 C00370 BC00370  +REFP EC00370
CALL JOB:SEARCH-R1-S13D
SET P028 P006
SFTON3D P028
SMOVL C00371 BC00371 V=166.7  +MOVJ EC00371
MOVL C00372 BC00372 V=1000.0  +MOVJ EC00372 VJ=100.00
'EndPath S4102
SFTOF3D
MOVJ C00373 BC00373 VJ=100.00  +MOVJ EC00373 VJ=100.00
SMOVL C00374 BC00374 V=166.7  +MOVJ EC00374
SREFP 3 C00375 BC00375  +REFP EC00375
CALL JOB:SEARCH-R1-S13D
SET P056 P006
SFTON3D P056
SMOVL C00376 BC00376 V=166.7  +MOVJ EC00376
SREFP 3 C00377 BC00377  +REFP EC00377
CALL JOB:SEARCH-R1-S13D
SET P056 P006
SFTON3D P056
SMOVL C00378 BC00378 V=166.7  +MOVJ EC00378
MOVJ C00379 BC00379 VJ=100.00  +MOVJ EC00379 VJ=100.00
'Path S4103
SFTOF3D
MOVJ C00380 BC00380 VJ=100.00  +MOVJ EC00380 VJ=100.00
MOVL C00381 BC00381 V=666.7  +MOVJ EC00381 VJ=100.00
SMOVL C00382 BC00382 V=166.7  +MOVJ EC00382
SREFP 3 C00383 BC00383  +REFP EC00383
CALL JOB:SEARCH-R1-S13D
SET P033 P006
SFTON3D P033
SMOVL C00384 BC00384 V=166.7  +MOVJ EC00384
SMOVL C00385 BC00385 V=166.7  +MOVJ EC00385
SREFP 3 C00386 BC00386  +REFP EC00386
CALL JOB:SEARCH-R1-S13D
SET P033 P006
SFTON3D P033
SMOVL C00387 BC00387 V=166.7  +MOVJ EC00387
SMOVL C00388 BC00388 V=166.7  +MOVJ EC00388
SMOVL C00389 BC00389 V=166.7  +MOVJ EC00389
SREFP 3 C00390 BC00390  +REFP EC00390
CALL JOB:SEARCH-R1-S13D
SET P033 P006
SFTON3D P033
SMOVL C00391 BC00391 V=166.7  +MOVJ EC00391
MOVL C00392 BC00392 V=1000.0  +MOVJ EC00392 VJ=100.00
'EndPath S4103
'Path S4104
SFTOF3D
MOVJ C00393 BC00393 VJ=100.00  +MOVJ EC00393 VJ=100.00
MOVL C00394 BC00394 V=666.7  +MOVJ EC00394 VJ=100.00
SMOVL C00395 BC00395 V=166.7  +MOVJ EC00395
SREFP 3 C00396 BC00396  +REFP EC00396
CALL JOB:SEARCH-R1-S13D
SET P027 P006
SFTON3D P027
SMOVL C00397 BC00397 V=250.0  +MOVJ EC00397
SMOVL C00398 BC00398 V=166.7  +MOVJ EC00398
SREFP 3 C00399 BC00399  +REFP EC00399
CALL JOB:SEARCH-R1-S13D
SET P027 P006
SFTON3D P027
SMOVL C00400 BC00400 V=166.7  +MOVJ EC00400
SMOVL C00401 BC00401 V=166.7  +MOVJ EC00401
SREFP 3 C00402 BC00402  +REFP EC00402
CALL JOB:SEARCH-R1-S13D
SET P027 P006
SFTON3D P027
SMOVL C00403 BC00403 V=166.7  +MOVJ EC00403
MOVL C00404 BC00404 V=1000.0  +MOVJ EC00404 VJ=100.00
'EndPath S4104
MOVJ C00405 BC00405 VJ=100.00  +MOVJ EC00405 VJ=100.00
'Path S4105
SFTOF3D
MOVJ C00406 BC00406 VJ=100.00  +MOVJ EC00406 VJ=100.00
MOVL C00407 BC00407 V=666.7  +MOVJ EC00407 VJ=100.00
SMOVL C00408 BC00408 V=166.7  +MOVJ EC00408
SREFP 3 C00409 BC00409  +REFP EC00409
CALL JOB:SEARCH-R1-S13D
SET P030 P006
SFTON3D P030
SMOVL C00410 BC00410 V=166.7  +MOVJ EC00410
SREFP 3 C00411 BC00411  +REFP EC00411
CALL JOB:SEARCH-R1-S13D
SET P030 P006
SFTON3D P030
SMOVL C00412 BC00412 V=166.7  +MOVJ EC00412
MOVL C00413 BC00413 V=1000.0  +MOVJ EC00413 VJ=100.00
'EndPath S4105
'Path S4106
SFTOF3D
MOVJ C00414 BC00414 VJ=100.00  +MOVJ EC00414 VJ=100.00
MOVL C00415 BC00415 V=666.7  +MOVJ EC00415 VJ=100.00
SMOVL C00416 BC00416 V=166.7  +MOVJ EC00416
SREFP 3 C00417 BC00417  +REFP EC00417
CALL JOB:SEARCH-R1-S13D
SET P031 P006
SFTON3D P031
SMOVL C00418 BC00418 V=166.7  +MOVJ EC00418
SREFP 3 C00419 BC00419  +REFP EC00419
CALL JOB:SEARCH-R1-S13D
SET P031 P006
SFTON3D P031
SMOVL C00420 BC00420 V=166.7  +MOVJ EC00420
SFTOF3D
MOVL C00421 BC00421 V=666.7  +MOVJ EC00421 VJ=100.00
SMOVL C00422 BC00422 V=166.7  +MOVJ EC00422
SREFP 3 C00423 BC00423  +REFP EC00423
CALL JOB:SEARCH-R1-S13D
SET P098 P006
SFTON3D P098
SMOVL C00424 BC00424 V=166.7  +MOVJ EC00424
SREFP 3 C00425 BC00425  +REFP EC00425
CALL JOB:SEARCH-R1-S13D
SET P098 P006
SFTON3D P098
SMOVL C00426 BC00426 V=166.7  +MOVJ EC00426
MOVL C00427 BC00427 V=1000.0  +MOVJ EC00427 VJ=100.00
'EndPath S4106
MOVJ C00428 BC00428 VJ=100.00  +MOVJ EC00428 VJ=100.00
'Path S4107
SFTOF3D
MOVJ C00429 BC00429 VJ=100.00  +MOVJ EC00429 VJ=100.00
MOVL C00430 BC00430 V=666.7  +MOVJ EC00430 VJ=100.00
SMOVL C00431 BC00431 V=166.7  +MOVJ EC00431
SREFP 3 C00432 BC00432  +REFP EC00432
CALL JOB:SEARCH-R1-S13D
SET P032 P006
SFTON3D P032
SMOVL C00433 BC00433 V=166.7  +MOVJ EC00433
SREFP 3 C00434 BC00434  +REFP EC00434
CALL JOB:SEARCH-R1-S13D
SET P032 P006
SFTON3D P032
SMOVL C00435 BC00435 V=166.7  +MOVJ EC00435
SMOVL C00436 BC00436 V=250.0  +MOVJ EC00436
SMOVL C00437 BC00437 V=166.7  +MOVJ EC00437
SREFP 3 C00438 BC00438  +REFP EC00438
CALL JOB:SEARCH-R1-S13D
SET P032 P006
SFTON3D P032
SMOVL C00439 BC00439 V=166.7  +MOVJ EC00439
MOVL C00440 BC00440 V=1000.0  +MOVJ EC00440 VJ=100.00
'EndPath S4107
'
MOVJ C00441 BC00441 VJ=100.00  +MOVJ EC00441 VJ=100.00
'Path S4208
SFTOF3D
MOVJ C00442 BC00442 VJ=100.00  +MOVJ EC00442 VJ=100.00
MOVL C00443 BC00443 V=666.7  +MOVJ EC00443 VJ=100.00
SMOVL C00444 BC00444 V=166.7  +MOVJ EC00444
SREFP 3 C00445 BC00445  +REFP EC00445
CALL JOB:SEARCH-R1-S13D
SET P052 P006
SFTON3D P052
SMOVL C00446 BC00446 V=166.7  +MOVJ EC00446
SREFP 3 C00447 BC00447  +REFP EC00447
CALL JOB:SEARCH-R1-S13D
SET P052 P006
SFTON3D P052
SMOVL C00448 BC00448 V=166.7  +MOVJ EC00448
SFTOF3D
MOVL C00449 BC00449 V=1000.0  +MOVJ EC00449 VJ=100.00
SMOVL C00450 BC00450 V=500.0  +MOVJ EC00450
SMOVL C00451 BC00451 V=166.7  +MOVJ EC00451
SREFP 3 C00452 BC00452  +REFP EC00452
CALL JOB:SEARCH-R1-S13D
SET P088 P006
SFTON3D P088
SMOVL C00453 BC00453 V=166.7  +MOVJ EC00453
SMOVL C00454 BC00454 V=166.7  +MOVJ EC00454
SMOVL C00455 BC00455 V=166.7  +MOVJ EC00455
SREFP 3 C00456 BC00456  +REFP EC00456
CALL JOB:SEARCH-R1-S13D
SET P088 P006
SFTON3D P088
SMOVL C00457 BC00457 V=333.3  +MOVJ EC00457
SMOVL C00458 BC00458 V=666.7  +MOVJ EC00458
SFTOF3D
'EndPath S4208
MOVJ C00459 BC00459 VJ=100.00  +MOVJ EC00459 VJ=100.00
'Path S4209
SFTOF3D
MOVJ C00460 BC00460 VJ=100.00  +MOVJ EC00460 VJ=100.00
MOVL C00461 BC00461 V=666.7  +MOVJ EC00461 VJ=100.00
SMOVL C00462 BC00462 V=166.7  +MOVJ EC00462
SREFP 3 C00463 BC00463  +REFP EC00463
CALL JOB:SEARCH-R1-S13D
SET P053 P006
SFTON3D P053
SMOVL C00464 BC00464 V=166.7  +MOVJ EC00464
SMOVL C00465 BC00465 V=166.7  +MOVJ EC00465
SREFP 3 C00466 BC00466  +REFP EC00466
CALL JOB:SEARCH-R1-S13D
SET P053 P006
SFTON3D P053
SMOVL C00467 BC00467 V=166.7  +MOVJ EC00467
MOVL C00468 BC00468 V=1000.0  +MOVJ EC00468 VJ=100.00
'EndPath S4209
*BP1
MOVJ C00469 BC00469 VJ=100.00  +MOVJ EC00469 VJ=100.00
'Path W4108
SFTOF3D
SFTON3D P033
MOVJ C00470 BC00470 VJ=100.00  +MOVJ EC00470 VJ=100.00
SMOVL C00471 BC00471 V=666.7  +MOVJ EC00471
SMOVL C00472 BC00472 V=166.7 PL=0  +MOVJ EC00472
MACRO1 MJ#(0) ARGF14
ARCON
SMOVL C00473 BC00473 V=9.2  +MOVJ EC00473
ARCOF
SMOVL C00474 BC00474 V=800.0  +MOVJ EC00474
SMOVL C00475 BC00475 V=1000.0  +MOVJ EC00475
SFTOF3D
'EndPath W4108
'Path W4109
SFTOF3D
MOVJ C00476 BC00476 VJ=100.00  +MOVJ EC00476 VJ=100.00
MOVJ C00477 BC00477 VJ=100.00  +MOVJ EC00477 VJ=100.00
'Path W4110
SFTOF3D
SFTON3D P033
MOVJ C00478 BC00478 VJ=100.00  +MOVJ EC00478 VJ=100.00
SMOVL C00479 BC00479 V=800.0  +MOVJ EC00479
SMOVL C00480 BC00480 V=133.3 PL=0  +MOVJ EC00480
MACRO1 MJ#(0) ARGF9
ARCON
SMOVL C00481 BC00481 V=11.7  +MOVJ EC00481
SMOVL C00482 BC00482 V=11.7  +MOVJ EC00482
SMOVL C00483 BC00483 V=11.7  +MOVJ EC00483
ARCOF
SMOVL C00484 BC00484 V=800.0  +MOVJ EC00484
SMOVL C00485 BC00485 V=1000.0  +MOVJ EC00485
SFTOF3D
'EndPath W4110
MOVJ C00486 BC00486 VJ=100.00  +MOVJ EC00486 VJ=100.00
'9
MOVJ C00487 BC00487 VJ=100.00  +MOVJ EC00487 VJ=100.00
'Path W4111
SFTOF3D
SFTON3D P026
MOVJ C00488 BC00488 VJ=100.00  +MOVJ EC00488 VJ=100.00
SMOVL C00489 BC00489 V=666.7  +MOVJ EC00489
SMOVL C00490 BC00490 V=166.7 PL=0  +MOVJ EC00490
MACRO1 MJ#(0) ARGF14
ARCON
SMOVL C00491 BC00491 V=9.2  +MOVJ EC00491
ARCOF
SMOVL C00492 BC00492 V=800.0  +MOVJ EC00492
SMOVL C00493 BC00493 V=1000.0  +MOVJ EC00493
SFTOF3D
'EndPath W4111
'Path W4112
SFTOF3D
SFTON3D P026
MOVJ C00494 BC00494 VJ=100.00  +MOVJ EC00494 VJ=100.00
SMOVL C00495 BC00495 V=800.0  +MOVJ EC00495
SMOVL C00496 BC00496 V=150.0 PL=0  +MOVJ EC00496
ARCON
SMOVL C00497 BC00497 V=11.7  +MOVJ EC00497
SMOVL C00498 BC00498 V=11.7  +MOVJ EC00498
SMOVL C00499 BC00499 V=11.7  +MOVJ EC00499
ARCOF
SMOVL C00500 BC00500 V=800.0  +MOVJ EC00500
SMOVL C00501 BC00501 V=1000.0  +MOVJ EC00501
SFTOF3D
MOVJ C00502 BC00502 VJ=100.00  +MOVJ EC00502 VJ=100.00
MOVJ C00503 BC00503 VJ=100.00  +MOVJ EC00503 VJ=100.00
'uwaga na podajnik
'Path W4114
SFTOF3D
SFTON3D P026
MOVJ C00504 BC00504 VJ=100.00  +MOVJ EC00504 VJ=100.00
SMOVL C00505 BC00505 V=800.0  +MOVJ EC00505
SMOVL C00506 BC00506 V=150.0 PL=0  +MOVJ EC00506
ARCON
SMOVL C00507 BC00507 V=11.7  +MOVJ EC00507
ARCOF
SMOVL C00508 BC00508 V=800.0  +MOVJ EC00508
SMOVL C00509 BC00509 V=1000.0  +MOVJ EC00509
SFTOF3D
'EndPath W4114
'brak dostepu offset drutu 1cm
'Path W4115
SFTOF3D
SFTON3D P026
MOVJ C00510 BC00510 VJ=100.00  +MOVJ EC00510 VJ=100.00
SMOVL C00511 BC00511 V=800.0  +MOVJ EC00511
SMOVL C00512 BC00512 V=150.0 PL=0  +MOVJ EC00512
ARCON
SMOVL C00513 BC00513 V=11.7  +MOVJ EC00513
ARCOF
SMOVL C00514 BC00514 V=800.0  +MOVJ EC00514
SMOVL C00515 BC00515 V=1000.0  +MOVJ EC00515
SFTOF3D
SFTON3D P081
MOVJ C00516 BC00516 VJ=100.00  +MOVJ EC00516 VJ=100.00
SMOVL C00517 BC00517 V=666.7  +MOVJ EC00517
SMOVL C00518 BC00518 V=166.7 PL=0  +MOVJ EC00518
MACRO1 MJ#(0) ARGF14
ARCON
SMOVL C00519 BC00519 V=9.2  +MOVJ EC00519
ARCOF
SMOVL C00520 BC00520 V=800.0  +MOVJ EC00520
SMOVL C00521 BC00521 V=1000.0  +MOVJ EC00521
SFTOF3D
'EndPath W4111
'Path W4112
SFTOF3D
SFTON3D P081
MOVJ C00522 BC00522 VJ=100.00  +MOVJ EC00522 VJ=100.00
SMOVL C00523 BC00523 V=800.0  +MOVJ EC00523
SMOVL C00524 BC00524 V=150.0 PL=0  +MOVJ EC00524
ARCON
SMOVL C00525 BC00525 V=11.7  +MOVJ EC00525
SMOVL C00526 BC00526 V=11.7  +MOVJ EC00526
SMOVL C00527 BC00527 V=11.7  +MOVJ EC00527
ARCOF
SMOVL C00528 BC00528 V=800.0  +MOVJ EC00528
SMOVL C00529 BC00529 V=1000.0  +MOVJ EC00529
SFTOF3D
MOVJ C00530 BC00530 VJ=100.00  +MOVJ EC00530 VJ=100.00
MOVJ C00531 BC00531 VJ=100.00  +MOVJ EC00531 VJ=100.00
'uwaga na podajnik
'Path W4114
SFTOF3D
SFTON3D P081
MOVJ C00532 BC00532 VJ=100.00  +MOVJ EC00532 VJ=100.00
SMOVL C00533 BC00533 V=800.0  +MOVJ EC00533
SMOVL C00534 BC00534 V=150.0 PL=0  +MOVJ EC00534
ARCON
SMOVL C00535 BC00535 V=11.7  +MOVJ EC00535
ARCOF
SMOVL C00536 BC00536 V=800.0  +MOVJ EC00536
SMOVL C00537 BC00537 V=1000.0  +MOVJ EC00537
SFTOF3D
'EndPath W4114
'brak dostepu offset drutu 1cm
'Path W4115
SFTOF3D
SFTON3D P081
MOVJ C00538 BC00538 VJ=100.00  +MOVJ EC00538 VJ=100.00
SMOVL C00539 BC00539 V=800.0  +MOVJ EC00539
SMOVL C00540 BC00540 V=150.0 PL=0  +MOVJ EC00540
ARCON
SMOVL C00541 BC00541 V=11.7  +MOVJ EC00541
ARCOF
SMOVL C00542 BC00542 V=800.0  +MOVJ EC00542
SMOVL C00543 BC00543 V=1000.0  +MOVJ EC00543
SFTOF3D
'EndPath W4115
MOVJ C00544 BC00544 VJ=100.00  +MOVJ EC00544 VJ=100.00
'10
'11
MOVJ C00545 BC00545 VJ=100.00  +MOVJ EC00545 VJ=100.00
'Path W4118
SFTOF3D
SFTON3D P055
MOVJ C00546 BC00546 VJ=100.00  +MOVJ EC00546 VJ=100.00
SMOVL C00547 BC00547 V=800.0  +MOVJ EC00547
SMOVL C00548 BC00548 V=666.7  +MOVJ EC00548
SMOVL C00549 BC00549 V=166.7 PL=0  +MOVJ EC00549
ARCON
SMOVL C00550 BC00550 V=9.2  +MOVJ EC00550
SFTON3D P049
SMOVL C00551 BC00551 V=9.2  +MOVJ EC00551
SMOVL C00552 BC00552 V=9.2  +MOVJ EC00552
SMOVL C00553 BC00553 V=9.2  +MOVJ EC00553
SFTON3D P025
SMOVL C00554 BC00554 V=9.2  +MOVJ EC00554
ARCOF
SMOVL C00555 BC00555 V=800.0  +MOVJ EC00555
SMOVL C00556 BC00556 V=1000.0  +MOVJ EC00556
SFTOF3D
'EndPath W4118
'brak dostepu offset drutu 1cm
MOVJ C00557 BC00557 VJ=100.00  +MOVJ EC00557 VJ=100.00
'Path W4117
SFTOF3D
SFTON3D P025
MOVJ C00558 BC00558 VJ=100.00  +MOVJ EC00558 VJ=100.00
SMOVL C00559 BC00559 V=800.0  +MOVJ EC00559
SMOVL C00560 BC00560 V=166.7 PL=0  +MOVJ EC00560
ARCON
SMOVL C00561 BC00561 V=10.0  +MOVJ EC00561
ARCOF
SMOVL C00562 BC00562 V=800.0  +MOVJ EC00562
SMOVL C00563 BC00563 V=1000.0  +MOVJ EC00563
SFTOF3D
'EndPath W4117
'12
MOVJ C00564 BC00564 VJ=100.00  +MOVJ EC00564 VJ=100.00
MOVJ C00565 BC00565 VJ=100.00  +MOVJ EC00565 VJ=100.00
'Path W4859
SFTOF3D
SFTON3D P073
MOVJ C00566 BC00566 VJ=100.00  +MOVJ EC00566 VJ=100.00
SMOVL C00567 BC00567 V=800.0  +MOVJ EC00567
SMOVL C00568 BC00568 V=150.0 PL=0  +MOVJ EC00568
ARCON
SWVON WEV#(16)
SMOVL C00569 BC00569 V=6.7  +MOVJ EC00569
SFTON3D P047
SMOVL C00570 BC00570 V=7.5  +MOVJ EC00570
ARCOF
SWVOF
SMOVL C00571 BC00571 V=333.3  +MOVJ EC00571
COMM SMOVL C00572 BC00572 V=333.3  +MOVJ EC00572
COMM SMOVL C00573 BC00573 V=333.3  +MOVJ EC00573
COMM SMOVL C00574 BC00574 V=166.7 PL=0  +MOVJ EC00574
COMM ARCON
COMM SMOVL C00575 BC00575 V=9.2  +MOVJ EC00575
COMM SMOVL C00576 BC00576 V=9.2  +MOVJ EC00576
COMM ARCOF
COMM SMOVL C00577 BC00577 V=800.0  +MOVJ EC00577
COMM SMOVL C00578 BC00578 V=1000.0  +MOVJ EC00578
SFTOF3D
'EndPath W4859
MOVJ C00579 BC00579 VJ=100.00  +MOVJ EC00579 VJ=100.00
MOVJ C00580 BC00580 VJ=100.00  +MOVJ EC00580 VJ=100.00
'Path W4119
SFTOF3D
SFTON3D P034
MOVJ C00581 BC00581 VJ=100.00  +MOVJ EC00581 VJ=100.00
SMOVL C00582 BC00582 V=800.0  +MOVJ EC00582
SMOVL C00583 BC00583 V=150.0 PL=0  +MOVJ EC00583
ARCON
SMOVL C00584 BC00584 V=10.0  +MOVJ EC00584
SMOVL C00585 BC00585 V=10.0  +MOVJ EC00585
SMOVL C00586 BC00586 V=10.0  +MOVJ EC00586
ARCOF
SMOVL C00587 BC00587 V=800.0  +MOVJ EC00587
SMOVL C00588 BC00588 V=1000.0  +MOVJ EC00588
SFTOF3D
'EndPath W4119
'Path W4210
SFTOF3D
SFTON3D P050
MOVJ C00589 BC00589 VJ=100.00  +MOVJ EC00589 VJ=100.00
SMOVL C00590 BC00590 V=800.0  +MOVJ EC00590
SMOVL C00591 BC00591 V=150.0 PL=0  +MOVJ EC00591
ARCON
SMOVL C00592 BC00592 V=11.7  +MOVJ EC00592
ARCOF
SMOVL C00593 BC00593 V=800.0  +MOVJ EC00593
SMOVL C00594 BC00594 V=1000.0  +MOVJ EC00594
SFTOF3D
'EndPath W4210
'Path W4211
SFTOF3D
SFTON3D P034
MOVJ C00595 BC00595 VJ=100.00  +MOVJ EC00595 VJ=100.00
SMOVL C00596 BC00596 V=800.0  +MOVJ EC00596
SMOVL C00597 BC00597 V=166.7 PL=0  +MOVJ EC00597
ARCON
SWVON WEV#(66)
SMOVL C00598 BC00598 V=9.2  +MOVJ EC00598
SMOVL C00599 BC00599 V=9.2  +MOVJ EC00599
SMOVL C00600 BC00600 V=9.2  +MOVJ EC00600
ARCOF
SWVOF
SMOVL C00601 BC00601 V=800.0  +MOVJ EC00601
SMOVL C00602 BC00602 V=1000.0  +MOVJ EC00602
MOVJ C00603 BC00603 VJ=30.00  +MOVJ EC00603 VJ=30.00
MOVJ C00604 BC00604 VJ=30.00  +MOVJ EC00604 VJ=30.00
SFTOF3D
MACRO1 MJ#(0) ARGF6
MOVJ C00605 BC00605 VJ=30.00  +MOVJ EC00605 VJ=30.00
SFTON3D P063
SMOVL C00606 BC00606 V=133.3  +MOVJ EC00606
ARCON
SMOVL C00607 BC00607 V=11.7  +MOVJ EC00607
SMOVL C00608 BC00608 V=11.7  +MOVJ EC00608
SMOVL C00609 BC00609 V=11.7  +MOVJ EC00609
SFTON3D P062
SMOVL C00610 BC00610 V=11.7  +MOVJ EC00610
SMOVL C00611 BC00611 V=11.7  +MOVJ EC00611
SFTON3D P061
SMOVL C00612 BC00612 V=11.0  +MOVJ EC00612
SMOVL C00613 BC00613 V=11.0  +MOVJ EC00613
ARCOF
SMOVL C00614 BC00614 V=250.0  +MOVJ EC00614
SFTOF3D
MOVJ C00615 BC00615 VJ=30.00  +MOVJ EC00615 VJ=30.00
MOVJ C00616 BC00616 VJ=30.00  +MOVJ EC00616 VJ=30.00
'EndPath W4211
'Path W4210
SFTOF3D
SFTON3D P054
MOVJ C00617 BC00617 VJ=100.00  +MOVJ EC00617 VJ=100.00
SMOVL C00618 BC00618 V=800.0  +MOVJ EC00618
SMOVL C00619 BC00619 V=150.0 PL=0  +MOVJ EC00619
MACRO1 MJ#(0) ARGF14
ARCON
SWVON WEV#(67)
SMOVL C00620 BC00620 V=10.0  +MOVJ EC00620
SMOVL C00621 BC00621 V=10.0  +MOVJ EC00621
ARCOF
SWVOF
SMOVL C00622 BC00622 V=800.0  +MOVJ EC00622
SMOVL C00623 BC00623 V=1000.0  +MOVJ EC00623
SFTOF3D
'EndPath W4210
'Path W4121
SFTOF3D
SFTON3D P028
MOVJ C00624 BC00624 VJ=100.00  +MOVJ EC00624 VJ=100.00
SMOVL C00625 BC00625 V=800.0  +MOVJ EC00625
SMOVL C00626 BC00626 V=150.0 PL=0  +MOVJ EC00626
ARCON
SMOVL C00627 BC00627 V=9.2  +MOVJ EC00627
SMOVL C00628 BC00628 V=9.2  +MOVJ EC00628
SFTON3D P056
SMOVL C00629 BC00629 V=9.2  +MOVJ EC00629
SMOVL C00630 BC00630 V=9.2  +MOVJ EC00630
ARCOF
SMOVL C00631 BC00631 V=800.0  +MOVJ EC00631
SMOVL C00632 BC00632 V=1000.0  +MOVJ EC00632
SFTOF3D
'EndPath W4121
'brak dostepu offset 5mm
MOVJ C00633 BC00633 VJ=100.00  +MOVJ EC00633 VJ=100.00
'Path W4122
SFTOF3D
SFTON3D P028
MOVJ C00634 BC00634 VJ=100.00  +MOVJ EC00634 VJ=100.00
SMOVL C00635 BC00635 V=800.0  +MOVJ EC00635
SMOVL C00636 BC00636 V=166.7 PL=0  +MOVJ EC00636
ARCON
SMOVL C00637 BC00637 V=11.7  +MOVJ EC00637
ARCOF
SMOVL C00638 BC00638 V=800.0  +MOVJ EC00638
SMOVL C00639 BC00639 V=1000.0  +MOVJ EC00639
SFTOF3D
'EndPath W4122
MOVJ C00640 BC00640 VJ=100.00  +MOVJ EC00640 VJ=100.00
'13
MOVJ C00641 BC00641 VJ=100.00  +MOVJ EC00641 VJ=100.00
'Path W4123
SFTOF3D
SFTON3D P030
MOVJ C00642 BC00642 VJ=100.00  +MOVJ EC00642 VJ=100.00
SMOVL C00643 BC00643 V=800.0  +MOVJ EC00643
SMOVL C00644 BC00644 V=150.0 PL=0  +MOVJ EC00644
SREFP 1 C00645 BC00645  +REFP EC00645
SREFP 2 C00646 BC00646  +REFP EC00646
MACRO1 MJ#(0) ARGF9
ARCON
SWVON WEV#(10)
SFTON3D P031
SMOVL C00647 BC00647 V=6.7  +MOVJ EC00647
SFTON3D P098
SMOVL C00648 BC00648 V=6.7  +MOVJ EC00648
SMOVL C00649 BC00649 V=6.7  +MOVJ EC00649
ARCOF
SWVOF
SMOVL C00650 BC00650 V=800.0  +MOVJ EC00650
SMOVL C00651 BC00651 V=1000.0  +MOVJ EC00651
SFTOF3D
'EndPath W4123
'14
'15-brak
'Path W4212
SFTOF3D
SFTON3D P052
MOVJ C00652 BC00652 VJ=100.00  +MOVJ EC00652 VJ=100.00
SMOVL C00653 BC00653 V=800.0  +MOVJ EC00653
SMOVL C00654 BC00654 V=150.0 PL=0  +MOVJ EC00654
ARCON
SMOVL C00655 BC00655 V=10.8  +MOVJ EC00655
SMOVL C00656 BC00656 V=10.8  +MOVJ EC00656
SMOVL C00657 BC00657 V=10.8  +MOVJ EC00657
ARCOF
SMOVL C00658 BC00658 V=800.0  +MOVJ EC00658
MACRO1 MJ#(0) ARGF6
SMOVL C00659 BC00659 V=333.3  +MOVJ EC00659
SFTOF3D
'DODAC SHIFT
SFTON3D P088
SMOVL C00660 BC00660 V=133.3  +MOVJ EC00660
ARCON
SMOVL C00661 BC00661 V=10.8  +MOVJ EC00661
ARCOF
SMOVL C00662 BC00662 V=250.0  +MOVJ EC00662
SMOVL C00663 BC00663 V=1000.0  +MOVJ EC00663
SFTOF3D
'EndPath W4212
'16
'Path W4213
SFTOF3D
SFTON3D P053
MOVJ C00664 BC00664 VJ=100.00  +MOVJ EC00664 VJ=100.00
SMOVL C00665 BC00665 V=800.0  +MOVJ EC00665
SMOVL C00666 BC00666 V=150.0 PL=0  +MOVJ EC00666
MACRO1 MJ#(0) ARGF9
ARCON
SMOVL C00667 BC00667 V=10.8  +MOVJ EC00667
SMOVL C00668 BC00668 V=10.8  +MOVJ EC00668
SMOVL C00669 BC00669 V=10.8  +MOVJ EC00669
ARCOF
SMOVL C00670 BC00670 V=800.0  +MOVJ EC00670
SMOVL C00671 BC00671 V=1000.0  +MOVJ EC00671
SFTOF3D
'EndPath W4213
'Path W4124
SFTOF3D
SFTON3D P029
MOVJ C00672 BC00672 VJ=100.00  +MOVJ EC00672 VJ=100.00
SMOVL C00673 BC00673 V=800.0  +MOVJ EC00673
SMOVL C00674 BC00674 V=166.7 PL=0  +MOVJ EC00674
MACRO1 MJ#(0) ARGF14
ARCON
SMOVL C00675 BC00675 V=10.0  +MOVJ EC00675
SFTON3D P039
SMOVL C00676 BC00676 V=10.0  +MOVJ EC00676
SMOVL C00677 BC00677 V=10.0  +MOVJ EC00677
ARCOF
SMOVL C00678 BC00678 V=800.0  +MOVJ EC00678
SMOVL C00679 BC00679 V=1000.0  +MOVJ EC00679
SFTOF3D
'EndPath W4124
MOVJ C00680 BC00680 VJ=100.00  +MOVJ EC00680 VJ=100.00
'Path W4125
SFTOF3D
SFTON3D P029
MOVJ C00681 BC00681 VJ=100.00  +MOVJ EC00681 VJ=100.00
SMOVL C00682 BC00682 V=800.0  +MOVJ EC00682
SMOVL C00683 BC00683 V=150.0 PL=0  +MOVJ EC00683
ARCON
SWVON WEV#(16)
SFTON3D P037
SMOVL C00684 BC00684 V=11.7  +MOVJ EC00684
SFTON3D P038
SMOVL C00685 BC00685 V=11.7  +MOVJ EC00685
ARCOF
SWVOF
SMOVL C00686 BC00686 V=800.0  +MOVJ EC00686
SMOVL C00687 BC00687 V=1000.0  +MOVJ EC00687
SFTOF3D
'EndPath W4125
MOVJ C00688 BC00688 VJ=100.00  +MOVJ EC00688 VJ=100.00
'Path W4126
SFTOF3D
SFTON3D P039
MOVJ C00689 BC00689 VJ=100.00  +MOVJ EC00689 VJ=100.00
SMOVL C00690 BC00690 V=800.0  +MOVJ EC00690
SMOVL C00691 BC00691 V=166.7 PL=0  +MOVJ EC00691
ARCON
SWVON WEV#(16)
SFTON3D P040
SMOVL C00692 BC00692 V=11.7  +MOVJ EC00692
SFTON3D P041
SMOVL C00693 BC00693 V=11.7  +MOVJ EC00693
ARCOF
SWVOF
SMOVL C00694 BC00694 V=800.0  +MOVJ EC00694
SMOVL C00695 BC00695 V=1000.0  +MOVJ EC00695
SFTOF3D
SFTON3D P080
MOVJ C00696 BC00696 VJ=100.00  +MOVJ EC00696 VJ=100.00
SMOVL C00697 BC00697 V=800.0  +MOVJ EC00697
SMOVL C00698 BC00698 V=166.7 PL=0  +MOVJ EC00698
MACRO1 MJ#(0) ARGF14
ARCON
SWVON WEV#(16)
SMOVL C00699 BC00699 V=10.0  +MOVJ EC00699
SFTON3D P044
SMOVL C00700 BC00700 V=10.0  +MOVJ EC00700
SMOVL C00701 BC00701 V=10.0  +MOVJ EC00701
ARCOF
SWVOF
SMOVL C00702 BC00702 V=800.0  +MOVJ EC00702
SMOVL C00703 BC00703 V=1000.0  +MOVJ EC00703
SFTOF3D
'EndPath W4124
MOVJ C00704 BC00704 VJ=100.00  +MOVJ EC00704 VJ=100.00
'Path W4125
SFTOF3D
SFTON3D P080
MOVJ C00705 BC00705 VJ=100.00  +MOVJ EC00705 VJ=100.00
SMOVL C00706 BC00706 V=800.0  +MOVJ EC00706
SMOVL C00707 BC00707 V=150.0 PL=0  +MOVJ EC00707
ARCON
SWVON WEV#(16)
SFTON3D P042
SMOVL C00708 BC00708 V=11.7  +MOVJ EC00708
SFTON3D P043
SMOVL C00709 BC00709 V=11.7  +MOVJ EC00709
ARCOF
SWVOF
SMOVL C00710 BC00710 V=800.0  +MOVJ EC00710
SMOVL C00711 BC00711 V=1000.0  +MOVJ EC00711
SFTOF3D
'EndPath W4125
MOVJ C00712 BC00712 VJ=100.00  +MOVJ EC00712 VJ=100.00
'Path W4126
SFTOF3D
SFTON3D P080
MOVJ C00713 BC00713 VJ=100.00  +MOVJ EC00713 VJ=100.00
SMOVL C00714 BC00714 V=800.0  +MOVJ EC00714
SMOVL C00715 BC00715 V=166.7 PL=0  +MOVJ EC00715
ARCON
SWVON WEV#(16)
SFTON3D P045
SMOVL C00716 BC00716 V=11.7  +MOVJ EC00716
SFTON3D P046
SMOVL C00717 BC00717 V=11.7  +MOVJ EC00717
ARCOF
SWVOF
SMOVL C00718 BC00718 V=800.0  +MOVJ EC00718
SMOVL C00719 BC00719 V=1000.0  +MOVJ EC00719
SFTOF3D
'EndPath W4126
MOVJ C00720 BC00720 VJ=100.00  +MOVJ EC00720 VJ=100.00
'17
'Path W4127
SFTOF3D
SFTON3D P027
MOVJ C00721 BC00721 VJ=100.00  +MOVJ EC00721 VJ=100.00
SMOVL C00722 BC00722 V=800.0  +MOVJ EC00722
SMOVL C00723 BC00723 V=150.0 PL=0  +MOVJ EC00723
ARCON
SMOVL C00724 BC00724 V=10.0  +MOVJ EC00724
ARCOF
SMOVL C00725 BC00725 V=800.0  +MOVJ EC00725
SMOVL C00726 BC00726 V=1000.0  +MOVJ EC00726
SFTOF3D
'EndPath W4127
'Path W4128
SFTOF3D
SFTON3D P027
MOVJ C00727 BC00727 VJ=100.00  +MOVJ EC00727 VJ=100.00
SMOVL C00728 BC00728 V=800.0  +MOVJ EC00728
SMOVL C00729 BC00729 V=150.0 PL=0  +MOVJ EC00729
ARCON
SMOVL C00730 BC00730 V=11.7  +MOVJ EC00730
ARCOF
SMOVL C00731 BC00731 V=800.0  +MOVJ EC00731
SMOVL C00732 BC00732 V=1000.0  +MOVJ EC00732
SFTOF3D
COMM 'EndPath W4128
COMM 'Path W4129
COMM SFTOF3D
COMM SFTON3D P027
COMM MOVJ C00733 BC00733 VJ=100.00  +MOVJ EC00733 VJ=100.00
COMM SMOVL C00734 BC00734 V=800.0  +MOVJ EC00734
COMM SMOVL C00735 BC00735 V=150.0 PL=0  +MOVJ EC00735
COMM SMOVL C00736 BC00736 V=16.7  +MOVJ EC00736
COMM ARCOF
COMM SMOVL C00737 BC00737 V=800.0  +MOVJ EC00737
COMM SMOVL C00738 BC00738 V=1000.0  +MOVJ EC00738
COMM SFTOF3D
COMM 'EndPath W4129
'18
MOVJ C00739 BC00739 VJ=100.00  +MOVJ EC00739 VJ=100.00
'Path W4130
SFTOF3D
SFTON3D P024
MOVJ C00740 BC00740 VJ=100.00  +MOVJ EC00740 VJ=100.00
SMOVL C00741 BC00741 V=800.0  +MOVJ EC00741
SMOVL C00742 BC00742 V=150.0 PL=0  +MOVJ EC00742
ARCON
SWVON WEV#(16)
SMOVL C00743 BC00743 V=9.2  +MOVJ EC00743
SFTON3D P105
SMOVL C00744 BC00744 V=9.2  +MOVJ EC00744
SMOVL C00745 BC00745 V=9.2  +MOVJ EC00745
SFTON3D P036
SMOVL C00746 BC00746 V=9.2  +MOVJ EC00746
SFTON3D P035
MOVL C00747 BC00747 V=7.5  +MOVJ EC00747 VJ=0.78
ARCOF
SWVOF
SMOVL C00748 BC00748 V=800.0  +MOVJ EC00748
SMOVL C00749 BC00749 V=1000.0  +MOVJ EC00749
SFTOF3D
'EndPath W4130
'Path W4860
SFTOF3D
SFTON3D P071
MOVJ C00750 BC00750 VJ=100.00  +MOVJ EC00750 VJ=100.00
SMOVL C00751 BC00751 V=800.0  +MOVJ EC00751
SMOVL C00752 BC00752 V=150.0 PL=0  +MOVJ EC00752
MACRO1 MJ#(0) ARGF9
ARCON
SWVON WEV#(16)
SMOVL C00753 BC00753 V=9.2  +MOVJ EC00753
SFTON3D P048
SMOVL C00754 BC00754 V=9.2  +MOVJ EC00754
SMOVL C00755 BC00755 V=9.2  +MOVJ EC00755
ARCOF
SWVOF
SMOVL C00756 BC00756 V=333.3  +MOVJ EC00756
COMM SMOVL C00757 BC00757 V=666.7  +MOVJ EC00757
COMM SMOVL C00758 BC00758 V=333.3  +MOVJ EC00758
COMM SMOVL C00759 BC00759 V=166.7 PL=0  +MOVJ EC00759
COMM ARCON
COMM SMOVL C00760 BC00760 V=9.2  +MOVJ EC00760
COMM SMOVL C00761 BC00761 V=9.2  +MOVJ EC00761
COMM ARCOF
COMM SMOVL C00762 BC00762 V=800.0  +MOVJ EC00762
COMM SMOVL C00763 BC00763 V=1000.0  +MOVJ EC00763
COMM SFTOF3D
COMM 'EndPath W4860
COMM '19
MOVJ C00764 BC00764 VJ=100.00  +MOVJ EC00764 VJ=100.00
'Path W4131
SFTOF3D
SFTON3D P023
MOVJ C00765 BC00765 VJ=100.00  +MOVJ EC00765 VJ=100.00
SMOVL C00766 BC00766 V=800.0  +MOVJ EC00766
SMOVL C00767 BC00767 V=166.7 PL=0  +MOVJ EC00767
MACRO1 MJ#(0) ARGF6
ARCON
SWVON WEV#(66)
SMOVL C00768 BC00768 V=7.5  +MOVJ EC00768
SMOVL C00769 BC00769 V=7.5  +MOVJ EC00769
SMOVL C00770 BC00770 V=7.5  +MOVJ EC00770
ARCOF
SWVOF
SMOVL C00771 BC00771 V=800.0  +MOVJ EC00771
SMOVL C00772 BC00772 V=1000.0  +MOVJ EC00772
SFTOF3D
'EndPath W4131
MOVJ C00773 BC00773 VJ=100.00  +MOVJ EC00773 VJ=100.00
'Path W4214
SFTOF3D
SFTON3D P089
MOVJ C00774 BC00774 VJ=100.00  +MOVJ EC00774 VJ=100.00
SMOVL C00775 BC00775 V=800.0  +MOVJ EC00775
SMOVL C00776 BC00776 V=150.0 PL=0  +MOVJ EC00776
MACRO1 MJ#(0) ARGF9
ARCON
SWVON WEV#(16)
SMOVL C00777 BC00777 V=9.2  +MOVJ EC00777
SFTON3D P050
SMOVL C00778 BC00778 V=9.2  +MOVJ EC00778
SMOVL C00779 BC00779 V=9.2  +MOVJ EC00779
ARCOF
SWVOF
SMOVL C00780 BC00780 V=800.0  +MOVJ EC00780
SMOVL C00781 BC00781 V=1000.0  +MOVJ EC00781
SFTOF3D
'EndPath W4214
'Path W4215
SFTOF3D
SFTON3D P051
MOVJ C00782 BC00782 VJ=100.00  +MOVJ EC00782 VJ=100.00
SMOVL C00783 BC00783 V=800.0  +MOVJ EC00783
SMOVL C00784 BC00784 V=150.0 PL=0  +MOVJ EC00784
MACRO1 MJ#(0) ARGF9
ARCON
SWVON WEV#(60)
SMOVL C00785 BC00785 V=7.5  +MOVJ EC00785
SMOVL C00786 BC00786 V=7.5  +MOVJ EC00786
SMOVL C00787 BC00787 V=7.5  +MOVJ EC00787
ARCOF
SWVOF
SMOVL C00788 BC00788 V=800.0  +MOVJ EC00788
SMOVL C00789 BC00789 V=1000.0  +MOVJ EC00789
SFTOF3D
'EndPath W4215
MOVJ C00790 BC00790 VJ=100.00  +MOVJ EC00790 VJ=100.00
'20
'offset 5mm
MOVJ C00791 BC00791 VJ=100.00  +MOVJ EC00791 VJ=100.00
MOVJ C00792 BC00792 VJ=100.00  +MOVJ EC00792 VJ=100.00
'Path W4132
SFTOF3D
SFTON3D P032
MOVJ C00793 BC00793 VJ=100.00  +MOVJ EC00793 VJ=100.00
SMOVL C00794 BC00794 V=800.0  +MOVJ EC00794
SMOVL C00795 BC00795 V=150.0 PL=0  +MOVJ EC00795
ARCON
SMOVL C00796 BC00796 V=10.0  +MOVJ EC00796
SMOVL C00797 BC00797 V=10.0  +MOVJ EC00797
ARCOF
SMOVL C00798 BC00798 V=800.0  +MOVJ EC00798
SMOVL C00799 BC00799 V=1000.0  +MOVJ EC00799
SFTOF3D
JUMP *FFF
'EndPath W4132
'Path W4133
SFTOF3D
SFTON3D P032
MOVJ C00800 BC00800 VJ=100.00  +MOVJ EC00800 VJ=100.00
SMOVL C00801 BC00801 V=800.0  +MOVJ EC00801
SMOVL C00802 BC00802 V=166.7 PL=0  +MOVJ EC00802
ARCON
SMOVL C00803 BC00803 V=10.0  +MOVJ EC00803
ARCOF
SMOVL C00804 BC00804 V=800.0  +MOVJ EC00804
SMOVL C00805 BC00805 V=1000.0  +MOVJ EC00805
SFTOF3D
'EndPath W4133
'Path W4134
SFTOF3D
SFTON3D P032
MOVJ C00806 BC00806 VJ=100.00  +MOVJ EC00806 VJ=100.00
SMOVL C00807 BC00807 V=800.0  +MOVJ EC00807
SMOVL C00808 BC00808 V=150.0 PL=0  +MOVJ EC00808
ARCON
SMOVL C00809 BC00809 V=10.0  +MOVJ EC00809
ARCOF
SMOVL C00810 BC00810 V=800.0  +MOVJ EC00810
*FFF
SMOVL C00811 BC00811 V=1000.0  +MOVJ EC00811
SFTOF3D
'EndPath W4134
'offset 5mm
MOVJ C00812 BC00812 VJ=100.00  +MOVJ EC00812 VJ=100.00
'Path W4135
SFTOF3D
SFTON3D P032
MOVJ C00813 BC00813 VJ=100.00  +MOVJ EC00813 VJ=100.00
SMOVL C00814 BC00814 V=800.0  +MOVJ EC00814
SMOVL C00815 BC00815 V=166.7 PL=0  +MOVJ EC00815
ARCON
SMOVL C00816 BC00816 V=10.0  +MOVJ EC00816
ARCOF
SMOVL C00817 BC00817 V=800.0  +MOVJ EC00817
SMOVL C00818 BC00818 V=1000.0  +MOVJ EC00818
SFTOF3D
'EndPath W4135
MOVJ C00819 BC00819 VJ=100.00  +MOVJ EC00819 VJ=100.00
'Path W4136
SFTOF3D
SFTON3D P032
MOVJ C00820 BC00820 VJ=100.00  +MOVJ EC00820 VJ=100.00
SMOVL C00821 BC00821 V=800.0  +MOVJ EC00821
SMOVL C00822 BC00822 V=166.7 PL=0  +MOVJ EC00822
ARCON
SMOVL C00823 BC00823 V=11.7  +MOVJ EC00823
SMOVL C00824 BC00824 V=11.7  +MOVJ EC00824
ARCOF
SMOVL C00825 BC00825 V=800.0  +MOVJ EC00825
SMOVL C00826 BC00826 V=1000.0  +MOVJ EC00826
SFTOF3D
'EndPath W4136
MOVJ C00827 BC00827 VJ=100.00  +MOVJ EC00827 VJ=100.00
MOVJ C00828 BC00828 VJ=100.00  +MOVJ EC00828 VJ=100.00
'Path W4137
SFTOF3D
SFTON3D P097
MACRO1 MJ#(0) ARGF9
MOVJ C00829 BC00829 VJ=100.00  +MOVJ EC00829 VJ=100.00
SMOVL C00830 BC00830 V=800.0  +MOVJ EC00830
SMOVL C00831 BC00831 V=166.7 PL=0  +MOVJ EC00831
ARCON
SMOVL C00832 BC00832 V=10.0  +MOVJ EC00832
SFTON3D P021
SMOVL C00833 BC00833 V=10.0  +MOVJ EC00833
SFTON3D P022
SMOVL C00834 BC00834 V=10.0  +MOVJ EC00834
SMOVL C00835 BC00835 V=10.0  +MOVJ EC00835
ARCOF
SMOVL C00836 BC00836 V=800.0  +MOVJ EC00836
SMOVL C00837 BC00837 V=1000.0  +MOVJ EC00837
SFTOF3D
'EndPath W4137
MOVJ C00838 BC00838 VJ=100.00  +MOVJ EC00838 VJ=100.00
'Path W4724
SFTOF3D
SFTON3D P095
MOVJ C00839 BC00839 VJ=100.00  +MOVJ EC00839 VJ=100.00
SMOVL C00840 BC00840 V=800.0  +MOVJ EC00840
SMOVL C00841 BC00841 V=150.0 PL=0  +MOVJ EC00841
ARCON
SMOVL C00842 BC00842 V=10.0  +MOVJ EC00842
SMOVL C00843 BC00843 V=10.0  +MOVJ EC00843
SMOVL C00844 BC00844 V=10.0  +MOVJ EC00844
ARCOF
SMOVL C00845 BC00845 V=800.0  +MOVJ EC00845
SMOVL C00846 BC00846 V=1000.0  +MOVJ EC00846
SFTOF3D
'EndPath W4724
'Path W4725
SFTOF3D
SFTON3D P096
MOVJ C00847 BC00847 VJ=100.00  +MOVJ EC00847 VJ=100.00
SMOVL C00848 BC00848 V=800.0  +MOVJ EC00848
SMOVL C00849 BC00849 V=150.0 PL=0  +MOVJ EC00849
ARCON
SMOVL C00850 BC00850 V=10.0  +MOVJ EC00850
SMOVL C00851 BC00851 V=10.0  +MOVJ EC00851
ARCOF
SMOVL C00852 BC00852 V=800.0  +MOVJ EC00852
SMOVL C00853 BC00853 V=1000.0  +MOVJ EC00853
SFTOF3D
'EndPath W4725
MOVJ C00854 BC00854 VJ=100.00  +MOVJ EC00854 VJ=100.00
'Path W4861
SFTOF3D
SFTON3D P071
MOVJ C00855 BC00855 VJ=100.00  +MOVJ EC00855 VJ=100.00
SMOVL C00856 BC00856 V=800.0  +MOVJ EC00856
SMOVL C00857 BC00857 V=150.0 PL=0  +MOVJ EC00857
MACRO1 MJ#(0) ARGF14
ARCON
SWVON WEV#(16)
SMOVL C00858 BC00858 V=9.2  +MOVJ EC00858
SFTON3D P073
SMOVL C00859 BC00859 V=9.2  +MOVJ EC00859
SMOVL C00860 BC00860 V=9.2  +MOVJ EC00860
ARCOF
SWVOF
SMOVL C00861 BC00861 V=800.0  +MOVJ EC00861
SMOVL C00862 BC00862 V=1000.0  +MOVJ EC00862
SFTOF3D
SMOVL C00863 BC00863 V=1000.0  +MOVJ EC00863
COMM SFTOF3D
COMM SFTON3D P080
COMM MOVJ C00864 BC00864 VJ=100.00  +MOVJ EC00864 VJ=100.00
COMM SMOVL C00865 BC00865 V=800.0  +MOVJ EC00865
COMM SMOVL C00866 BC00866 V=150.0 PL=0  +MOVJ EC00866
COMM MACRO1 MJ#(0) ARGF14
COMM ARCON
COMM SMOVL C00867 BC00867 V=9.2  +MOVJ EC00867
COMM SFTON3D P080
COMM SMOVL C00868 BC00868 V=9.2  +MOVJ EC00868
COMM SMOVL C00869 BC00869 V=9.2  +MOVJ EC00869
COMM ARCOF
COMM SMOVL C00870 BC00870 V=800.0  +MOVJ EC00870
COMM SMOVL C00871 BC00871 V=1000.0  +MOVJ EC00871
SFTOF3D
'EndPath W4861
MOVJ C00872 BC00872 VJ=100.00  +MOVJ EC00872 VJ=100.00
MOVJ C00873 BC00873 VJ=100.00  +MOVJ EC00873 VJ=100.00
MOVJ C00874 BC00874 VJ=100.00  +MOVJ EC00874 VJ=100.00
MOVJ C00875 BC00875 VJ=100.00  +MOVJ EC00875 VJ=100.00
MOVJ C00876 BC00876 VJ=100.00  +MOVJ EC00876 VJ=100.00
MOVJ C00877 BC00877 VJ=100.00  +MOVJ EC00877 VJ=100.00
MOVL C00878 BC00878 V=1000.0  +MOVJ EC00878 VJ=100.00
SFTON3D P048
MOVL C00879 BC00879 V=166.7 PL=0  +MOVJ EC00879 VJ=100.00
ARCON
SMOVL C00880 BC00880 V=9.2  +MOVJ EC00880
SFTON3D P047
SMOVL C00881 BC00881 V=9.2  +MOVJ EC00881
SMOVL C00882 BC00882 V=9.2  +MOVJ EC00882
ARCOF
MOVL C00883 BC00883 V=666.7  +MOVJ EC00883 VJ=100.00
SFTOF3D
MOVJ C00884 BC00884 VJ=100.00  +MOVJ EC00884 VJ=100.00
CALL JOB:CLEAN-R1_KM_3P
'cut_wire_dol
'cut_wire_dol
'cut_wire_dol
MOVJ C00885 BC00885 VJ=100.00  +MOVJ EC00885 VJ=100.00
MOVJ C00886 BC00886 VJ=100.00  +MOVJ EC00886 VJ=100.00
MOVJ C00887 BC00887 VJ=100.00  +MOVJ EC00887 VJ=100.00
'Path S4138
SFTOF3D
MOVJ C00888 BC00888 VJ=100.00  +MOVJ EC00888 VJ=100.00
MOVL C00889 BC00889 V=800.0  +MOVJ EC00889 VJ=100.00
SMOVL C00890 BC00890 V=166.7  +MOVJ EC00890
SREFP 3 C00891 BC00891  +REFP EC00891
CALL JOB:SEARCH-R1-S13D
SET P049 P006
SFTON3D P049
SMOVL C00892 BC00892 V=166.7  +MOVJ EC00892
SMOVL C00893 BC00893 V=166.7  +MOVJ EC00893
SREFP 3 C00894 BC00894  +REFP EC00894
CALL JOB:SEARCH-R1-S13D
SET P049 P006
SFTON3D P049
SMOVL C00895 BC00895 V=166.7  +MOVJ EC00895
MOVL C00896 BC00896 V=800.0  +MOVJ EC00896 VJ=100.00
MOVL C00897 BC00897 V=1000.0  +MOVJ EC00897 VJ=100.00
'EndPath S4138
'Path S4139
SFTOF3D
MOVJ C00898 BC00898 VJ=100.00  +MOVJ EC00898 VJ=100.00
MOVL C00899 BC00899 V=800.0  +MOVJ EC00899 VJ=100.00
SMOVL C00900 BC00900 V=166.7  +MOVJ EC00900
SREFP 3 C00901 BC00901  +REFP EC00901
CALL JOB:SEARCH-R1-S13D
SET P048 P006
SFTON3D P048
SMOVL C00902 BC00902 V=166.7  +MOVJ EC00902
SMOVL C00903 BC00903 V=166.7  +MOVJ EC00903
SREFP 3 C00904 BC00904  +REFP EC00904
CALL JOB:SEARCH-R1-S13D
SET P048 P006
SFTON3D P048
SMOVL C00905 BC00905 V=166.7  +MOVJ EC00905
MOVL C00906 BC00906 V=800.0  +MOVJ EC00906 VJ=100.00
MOVL C00907 BC00907 V=1000.0  +MOVJ EC00907 VJ=100.00
'EndPath S4139
'Path S4140
SFTOF3D
MOVJ C00908 BC00908 VJ=100.00  +MOVJ EC00908 VJ=100.00
MOVL C00909 BC00909 V=800.0  +MOVJ EC00909 VJ=100.00
SMOVL C00910 BC00910 V=166.7  +MOVJ EC00910
SREFP 3 C00911 BC00911  +REFP EC00911
CALL JOB:SEARCH-R1-S13D
SET P047 P006
SFTON3D P047
SMOVL C00912 BC00912 V=166.7  +MOVJ EC00912
SMOVL C00913 BC00913 V=166.7  +MOVJ EC00913
SREFP 3 C00914 BC00914  +REFP EC00914
CALL JOB:SEARCH-R1-S13D
SET P047 P006
SFTON3D P047
SMOVL C00915 BC00915 V=166.7  +MOVJ EC00915
MOVL C00916 BC00916 V=800.0  +MOVJ EC00916 VJ=100.00
MOVL C00917 BC00917 V=1000.0  +MOVJ EC00917 VJ=100.00
'EndPath S4140
MOVJ C00918 BC00918 VJ=100.00  +MOVJ EC00918 VJ=100.00
MOVJ C00919 BC00919 VJ=100.00  +MOVJ EC00919 VJ=100.00
MOVJ C00920 BC00920 VJ=100.00  +MOVJ EC00920 VJ=100.00
MOVJ C00921 BC00921 VJ=100.00  +MOVJ EC00921 VJ=100.00
'Path S4141
SFTOF3D
MOVJ C00922 BC00922 VJ=100.00  +MOVJ EC00922 VJ=100.00
MOVL C00923 BC00923 V=800.0  +MOVJ EC00923 VJ=100.00
SMOVL C00924 BC00924 V=166.7  +MOVJ EC00924
SREFP 3 C00925 BC00925  +REFP EC00925
CALL JOB:SEARCH-R1-S13D
SET P046 P006
SFTON3D P046
SMOVL C00926 BC00926 V=166.7  +MOVJ EC00926
SMOVL C00927 BC00927 V=166.7  +MOVJ EC00927
SREFP 3 C00928 BC00928  +REFP EC00928
CALL JOB:SEARCH-R1-S13D
SET P046 P006
SFTON3D P046
SMOVL C00929 BC00929 V=166.7  +MOVJ EC00929
MOVL C00930 BC00930 V=1000.0  +MOVJ EC00930 VJ=100.00
'EndPath S4141
'Path S4142
SFTOF3D
MOVJ C00931 BC00931 VJ=100.00  +MOVJ EC00931 VJ=100.00
MOVL C00932 BC00932 V=800.0  +MOVJ EC00932 VJ=100.00
SMOVL C00933 BC00933 V=166.7  +MOVJ EC00933
SREFP 3 C00934 BC00934  +REFP EC00934
CALL JOB:SEARCH-R1-S13D
SET P045 P006
SFTON3D P045
SMOVL C00935 BC00935 V=166.7  +MOVJ EC00935
SMOVL C00936 BC00936 V=166.7  +MOVJ EC00936
SREFP 3 C00937 BC00937  +REFP EC00937
CALL JOB:SEARCH-R1-S13D
SET P045 P006
SFTON3D P045
SMOVL C00938 BC00938 V=166.7  +MOVJ EC00938
MOVL C00939 BC00939 V=1000.0  +MOVJ EC00939 VJ=100.00
'EndPath S4142
'Path S4143
SFTOF3D
MOVJ C00940 BC00940 VJ=100.00  +MOVJ EC00940 VJ=100.00
MOVL C00941 BC00941 V=800.0  +MOVJ EC00941 VJ=100.00
SMOVL C00942 BC00942 V=166.7  +MOVJ EC00942
SREFP 3 C00943 BC00943  +REFP EC00943
CALL JOB:SEARCH-R1-S13D
SET P044 P006
SFTON3D P044
SMOVL C00944 BC00944 V=166.7  +MOVJ EC00944
SMOVL C00945 BC00945 V=166.7  +MOVJ EC00945
SREFP 3 C00946 BC00946  +REFP EC00946
CALL JOB:SEARCH-R1-S13D
SET P044 P006
SFTON3D P044
SMOVL C00947 BC00947 V=166.7  +MOVJ EC00947
MOVL C00948 BC00948 V=1000.0  +MOVJ EC00948 VJ=100.00
'EndPath S4143
MOVJ C00949 BC00949 VJ=100.00  +MOVJ EC00949 VJ=100.00
MOVJ C00950 BC00950 VJ=100.00  +MOVJ EC00950 VJ=100.00
'Path S4144
SFTOF3D
MOVJ C00951 BC00951 VJ=100.00  +MOVJ EC00951 VJ=100.00
MOVL C00952 BC00952 V=800.0  +MOVJ EC00952 VJ=100.00
SMOVL C00953 BC00953 V=166.7  +MOVJ EC00953
SREFP 3 C00954 BC00954  +REFP EC00954
CALL JOB:SEARCH-R1-S13D
SET P043 P006
SFTON3D P043
SMOVL C00955 BC00955 V=166.7  +MOVJ EC00955
SMOVL C00956 BC00956 V=166.7  +MOVJ EC00956
SREFP 3 C00957 BC00957  +REFP EC00957
CALL JOB:SEARCH-R1-S13D
SET P043 P006
SFTON3D P043
SMOVL C00958 BC00958 V=166.7  +MOVJ EC00958
MOVL C00959 BC00959 V=1000.0  +MOVJ EC00959 VJ=100.00
'EndPath S4144
'Path S4145
SFTOF3D
MOVJ C00960 BC00960 VJ=100.00  +MOVJ EC00960 VJ=100.00
MOVL C00961 BC00961 V=800.0  +MOVJ EC00961 VJ=100.00
SMOVL C00962 BC00962 V=166.7  +MOVJ EC00962
SREFP 3 C00963 BC00963  +REFP EC00963
CALL JOB:SEARCH-R1-S13D
SET P042 P006
SFTON3D P042
SMOVL C00964 BC00964 V=166.7  +MOVJ EC00964
SMOVL C00965 BC00965 V=166.7  +MOVJ EC00965
SREFP 3 C00966 BC00966  +REFP EC00966
CALL JOB:SEARCH-R1-S13D
SET P042 P006
SFTON3D P042
SMOVL C00967 BC00967 V=166.7  +MOVJ EC00967
MOVL C00968 BC00968 V=1000.0  +MOVJ EC00968 VJ=100.00
'EndPath S4145
'Path S4146
SFTOF3D
MOVJ C00969 BC00969 VJ=100.00  +MOVJ EC00969 VJ=100.00
MOVL C00970 BC00970 V=666.7  +MOVJ EC00970 VJ=100.00
SMOVL C00971 BC00971 V=166.7  +MOVJ EC00971
SREFP 3 C00972 BC00972  +REFP EC00972
CALL JOB:SEARCH-R1-S13D
SET P041 P006
SFTON3D P041
SMOVL C00973 BC00973 V=250.0  +MOVJ EC00973
SMOVL C00974 BC00974 V=166.7  +MOVJ EC00974
SREFP 3 C00975 BC00975  +REFP EC00975
CALL JOB:SEARCH-R1-S13D
SET P041 P006
SFTON3D P041
SMOVL C00976 BC00976 V=166.7  +MOVJ EC00976
SMOVL C00977 BC00977 V=166.7  +MOVJ EC00977
SREFP 3 C00978 BC00978  +REFP EC00978
CALL JOB:SEARCH-R1-S13D
SET P041 P006
SFTON3D P041
SMOVL C00979 BC00979 V=166.7  +MOVJ EC00979
MOVL C00980 BC00980 V=1000.0  +MOVJ EC00980 VJ=100.00
'EndPath S4146
'Path S4147
SFTOF3D
MOVJ C00981 BC00981 VJ=100.00  +MOVJ EC00981 VJ=100.00
SMOVL C00982 BC00982 V=666.7  +MOVJ EC00982
SMOVL C00983 BC00983 V=166.7  +MOVJ EC00983
SREFP 3 C00984 BC00984  +REFP EC00984
CALL JOB:SEARCH-R1-S13D
SET P040 P006
SFTON3D P040
SMOVL C00985 BC00985 V=166.7  +MOVJ EC00985
SMOVL C00986 BC00986 V=800.0  +MOVJ EC00986
SMOVL C00987 BC00987 V=166.7  +MOVJ EC00987
SREFP 3 C00988 BC00988  +REFP EC00988
CALL JOB:SEARCH-R1-S13D
SET P040 P006
SFTON3D P040
SMOVL C00989 BC00989 V=166.7  +MOVJ EC00989
SMOVL C00990 BC00990 V=166.7  +MOVJ EC00990
SREFP 3 C00991 BC00991  +REFP EC00991
CALL JOB:SEARCH-R1-S13D
SET P040 P006
SFTON3D P040
SMOVL C00992 BC00992 V=166.7  +MOVJ EC00992
MOVL C00993 BC00993 V=1000.0  +MOVJ EC00993 VJ=100.00
'EndPath S4147
'Path W4148
SFTOF3D
SFTON3D P040
MOVJ C00994 BC00994 VJ=100.00  +MOVJ EC00994 VJ=100.00
SMOVL C00995 BC00995 V=800.0  +MOVJ EC00995
SMOVL C00996 BC00996 V=150.0 PL=0  +MOVJ EC00996
ARCON
SMOVL C00997 BC00997 V=10.0  +MOVJ EC00997
ARCOF
SMOVL C00998 BC00998 V=800.0  +MOVJ EC00998
SMOVL C00999 BC00999 V=1000.0  +MOVJ EC00999
SFTOF3D
'EndPath W4148
'Path W4149
SFTOF3D
SFTON3D P040
MOVJ C01000 BC01000 VJ=100.00  +MOVJ EC01000 VJ=100.00
SMOVL C01001 BC01001 V=800.0  +MOVJ EC01001
SMOVL C01002 BC01002 V=150.0 PL=0  +MOVJ EC01002
COMM ARCON
COMM SMOVL C01003 BC01003 V=11.7  +MOVJ EC01003
COMM ARCOF
SMOVL C01004 BC01004 V=800.0  +MOVJ EC01004
SMOVL C01005 BC01005 V=1000.0  +MOVJ EC01005
SFTOF3D
'EndPath W4149
'Path W4150
SFTOF3D
SFTON3D P040
COMM MOVJ C01006 BC01006 VJ=15.00  +MOVJ EC01006 VJ=15.00
COMM MOVJ C01007 BC01007 VJ=100.00  +MOVJ EC01007 VJ=100.00
COMM SMOVL C01008 BC01008 V=800.0  +MOVJ EC01008
COMM SMOVL C01009 BC01009 V=150.0 PL=0  +MOVJ EC01009
COMM ARCON
COMM SMOVL C01010 BC01010 V=11.7  +MOVJ EC01010
COMM ARCOF
COMM SMOVL C01011 BC01011 V=800.0  +MOVJ EC01011
COMM SMOVL C01012 BC01012 V=1000.0  +MOVJ EC01012
SFTOF3D
'EndPath W4150
'
MOVJ C01013 BC01013 VJ=100.00  +MOVJ EC01013 VJ=100.00
MOVJ C01014 BC01014 VJ=100.00  +MOVJ EC01014 VJ=100.00
'Path W4151
SFTOF3D
SFTON3D P045
MOVJ C01015 BC01015 VJ=100.00  +MOVJ EC01015 VJ=100.00
SMOVL C01016 BC01016 V=800.0  +MOVJ EC01016
SMOVL C01017 BC01017 V=150.0 PL=0  +MOVJ EC01017
MACRO1 MJ#(0) ARGF9
ARCON
SMOVL C01018 BC01018 V=11.7  +MOVJ EC01018
ARCOF
SMOVL C01019 BC01019 V=800.0  +MOVJ EC01019
SMOVL C01020 BC01020 V=1000.0  +MOVJ EC01020
SFTOF3D
'EndPath W4151
'Path W4152
SFTOF3D
SFTON3D P044
MOVJ C01021 BC01021 VJ=100.00  +MOVJ EC01021 VJ=100.00
SMOVL C01022 BC01022 V=800.0  +MOVJ EC01022
SMOVL C01023 BC01023 V=166.7 PL=0  +MOVJ EC01023
ARCON
SMOVL C01024 BC01024 V=11.7  +MOVJ EC01024
ARCOF
SMOVL C01025 BC01025 V=800.0  +MOVJ EC01025
SMOVL C01026 BC01026 V=1000.0  +MOVJ EC01026
SFTOF3D
'EndPath W4152
'Path W4153
SFTOF3D
SFTON3D P046
MOVJ C01027 BC01027 VJ=100.00  +MOVJ EC01027 VJ=100.00
SMOVL C01028 BC01028 V=800.0  +MOVJ EC01028
SMOVL C01029 BC01029 V=166.7 PL=0  +MOVJ EC01029
MACRO1 MJ#(0) ARGF14
ARCON
SMOVL C01030 BC01030 V=10.0  +MOVJ EC01030
SMOVL C01031 BC01031 V=10.0  +MOVJ EC01031
ARCOF
SMOVL C01032 BC01032 V=800.0  +MOVJ EC01032
SMOVL C01033 BC01033 V=1000.0  +MOVJ EC01033
SFTOF3D
'EndPath W4153
MOVJ C01034 BC01034 VJ=100.00  +MOVJ EC01034 VJ=100.00
MOVJ C01035 BC01035 VJ=100.00  +MOVJ EC01035 VJ=100.00
MOVJ C01036 BC01036 VJ=100.00  +MOVJ EC01036 VJ=100.00
MOVJ C01037 BC01037 VJ=100.00  +MOVJ EC01037 VJ=100.00
'1
'uwaga na podajnik
'Path W4154
SFTOF3D
SFTON3D P048
MOVJ C01038 BC01038 VJ=100.00  +MOVJ EC01038 VJ=100.00
SMOVL C01039 BC01039 V=800.0  +MOVJ EC01039
SMOVL C01040 BC01040 V=150.0 PL=0  +MOVJ EC01040
ARCON
SMOVL C01041 BC01041 V=10.0  +MOVJ EC01041
ARCOF
SMOVL C01042 BC01042 V=800.0  +MOVJ EC01042
SMOVL C01043 BC01043 V=1000.0  +MOVJ EC01043
SFTOF3D
'EndPath W4154
'Path W4155
SFTOF3D
SFTON3D P049
MOVJ C01044 BC01044 VJ=100.00  +MOVJ EC01044 VJ=100.00
SMOVL C01045 BC01045 V=800.0  +MOVJ EC01045
SMOVL C01046 BC01046 V=150.0 PL=0  +MOVJ EC01046
MACRO1 MJ#(0) ARGF6
ARCON
SMOVL C01047 BC01047 V=9.2  +MOVJ EC01047
SMOVL C01048 BC01048 V=9.2  +MOVJ EC01048
SMOVL C01049 BC01049 V=9.2  +MOVJ EC01049
SMOVL C01050 BC01050 V=9.2  +MOVJ EC01050
SMOVL C01051 BC01051 V=9.2  +MOVJ EC01051
ARCOF
SMOVL C01052 BC01052 V=800.0  +MOVJ EC01052
SMOVL C01053 BC01053 V=500.0  +MOVJ EC01053
SMOVL C01054 BC01054 V=133.3  +MOVJ EC01054
ARCON
SMOVL C01055 BC01055 V=13.3  +MOVJ EC01055
ARCOF
SMOVL C01056 BC01056 V=166.7  +MOVJ EC01056
ARCON
SMOVL C01057 BC01057 V=10.0  +MOVJ EC01057
ARCOF
SMOVL C01058 BC01058 V=250.0  +MOVJ EC01058
SMOVL C01059 BC01059 V=500.0  +MOVJ EC01059
SMOVL C01060 BC01060 V=500.0  +MOVJ EC01060
SMOVL C01061 BC01061 V=500.0  +MOVJ EC01061
SMOVL C01062 BC01062 V=133.3  +MOVJ EC01062
ARCON
SMOVL C01063 BC01063 V=13.3  +MOVJ EC01063
ARCOF
SMOVL C01064 BC01064 V=166.7  +MOVJ EC01064
SMOVL C01065 BC01065 V=166.7  +MOVJ EC01065
ARCON
SMOVL C01066 BC01066 V=10.0  +MOVJ EC01066
ARCOF
SMOVL C01067 BC01067 V=800.0  +MOVJ EC01067
SFTOF3D
'EndPath W4155
MOVJ C01068 BC01068 VJ=100.00  +MOVJ EC01068 VJ=100.00
MOVJ C01069 BC01069 VJ=100.00  +MOVJ EC01069 VJ=100.00
MOVJ C01070 BC01070 VJ=100.00  +MOVJ EC01070 VJ=100.00
MOVJ C01071 BC01071 VJ=100.00  +MOVJ EC01071 VJ=100.00
'2
'Path W4156
SFTOF3D
SFTON3D P043
MOVJ C01072 BC01072 VJ=100.00  +MOVJ EC01072 VJ=100.00
SMOVL C01073 BC01073 V=800.0  +MOVJ EC01073
SMOVL C01074 BC01074 V=166.7 PL=0  +MOVJ EC01074
MACRO1 MJ#(0) ARGF9
ARCON
SMOVL C01075 BC01075 V=11.7  +MOVJ EC01075
ARCOF
SMOVL C01076 BC01076 V=800.0  +MOVJ EC01076
SMOVL C01077 BC01077 V=1000.0  +MOVJ EC01077
SFTOF3D
'EndPath W4156
'Path W4157
SFTOF3D
SFTON3D P042
MOVJ C01078 BC01078 VJ=100.00  +MOVJ EC01078 VJ=100.00
SMOVL C01079 BC01079 V=800.0  +MOVJ EC01079
SMOVL C01080 BC01080 V=150.0 PL=0  +MOVJ EC01080
ARCON
SMOVL C01081 BC01081 V=11.7  +MOVJ EC01081
ARCOF
SMOVL C01082 BC01082 V=800.0  +MOVJ EC01082
SMOVL C01083 BC01083 V=1000.0  +MOVJ EC01083
SFTOF3D
'EndPath W4157
'3
MOVJ C01084 BC01084 VJ=100.00  +MOVJ EC01084 VJ=100.00
MOVJ C01085 BC01085 VJ=100.00  +MOVJ EC01085 VJ=100.00
MOVJ C01086 BC01086 VJ=100.00  +MOVJ EC01086 VJ=100.00
MOVJ C01087 BC01087 VJ=100.00  +MOVJ EC01087 VJ=100.00
'Path W4158
SFTOF3D
SFTON3D P047
MOVJ C01088 BC01088 VJ=100.00  +MOVJ EC01088 VJ=100.00
SMOVL C01089 BC01089 V=800.0  +MOVJ EC01089
SMOVL C01090 BC01090 V=150.0 PL=0  +MOVJ EC01090
ARCON
SMOVL C01091 BC01091 V=11.7  +MOVJ EC01091
ARCOF
SMOVL C01092 BC01092 V=800.0  +MOVJ EC01092
SMOVL C01093 BC01093 V=1000.0  +MOVJ EC01093
SFTOF3D
'EndPath W4158
'Path W4159
SFTOF3D
SFTON3D P047
MOVJ C01094 BC01094 VJ=100.00  +MOVJ EC01094 VJ=100.00
SMOVL C01095 BC01095 V=800.0  +MOVJ EC01095
SMOVL C01096 BC01096 V=150.0 PL=0  +MOVJ EC01096
ARCON
SMOVL C01097 BC01097 V=11.7  +MOVJ EC01097
ARCOF
SMOVL C01098 BC01098 V=800.0  +MOVJ EC01098
SMOVL C01099 BC01099 V=1000.0  +MOVJ EC01099
SFTOF3D
'EndPath W4159
MOVJ C01100 BC01100 VJ=100.00  +MOVJ EC01100 VJ=100.00
MOVJ C01101 BC01101 VJ=100.00  +MOVJ EC01101 VJ=100.00
MOVJ C01102 BC01102 VJ=100.00  +MOVJ EC01102 VJ=100.00
MOVJ C01103 BC01103 VJ=100.00  +MOVJ EC01103 VJ=100.00
'Path W4160
SFTOF3D
SFTON3D P043
MOVJ C01104 BC01104 VJ=100.00  +MOVJ EC01104 VJ=100.00
SMOVL C01105 BC01105 V=800.0  +MOVJ EC01105
SMOVL C01106 BC01106 V=150.0 PL=0  +MOVJ EC01106
ARCON
SMOVL C01107 BC01107 V=11.7  +MOVJ EC01107
ARCOF
SMOVL C01108 BC01108 V=800.0  +MOVJ EC01108
SMOVL C01109 BC01109 V=1000.0  +MOVJ EC01109
SFTOF3D
'EndPath W4160
'Path W4161
SFTOF3D
SFTON3D P042
MOVJ C01110 BC01110 VJ=100.00  +MOVJ EC01110 VJ=100.00
SMOVL C01111 BC01111 V=800.0  +MOVJ EC01111
SMOVL C01112 BC01112 V=166.7 PL=0  +MOVJ EC01112
ARCON
SMOVL C01113 BC01113 V=11.7  +MOVJ EC01113
ARCOF
SMOVL C01114 BC01114 V=800.0  +MOVJ EC01114
SMOVL C01115 BC01115 V=1000.0  +MOVJ EC01115
SFTOF3D
'EndPath W4161
MOVJ C01116 BC01116 VJ=100.00  +MOVJ EC01116 VJ=100.00
'Path W4162
SFTOF3D
SFTON3D P046
MOVJ C01117 BC01117 VJ=100.00  +MOVJ EC01117 VJ=100.00
SMOVL C01118 BC01118 V=800.0  +MOVJ EC01118
SMOVL C01119 BC01119 V=166.7 PL=0  +MOVJ EC01119
MACRO1 MJ#(0) ARGF14
ARCON
SMOVL C01120 BC01120 V=10.0  +MOVJ EC01120
ARCOF
SMOVL C01121 BC01121 V=800.0  +MOVJ EC01121
SMOVL C01122 BC01122 V=1000.0  +MOVJ EC01122
SFTOF3D
'EndPath W4162
'Path W4163
SFTOF3D
SFTON3D P044
MOVJ C01123 BC01123 VJ=100.00  +MOVJ EC01123 VJ=100.00
SMOVL C01124 BC01124 V=800.0  +MOVJ EC01124
SMOVL C01125 BC01125 V=150.0 PL=0  +MOVJ EC01125
MACRO1 MJ#(0) ARGF9
ARCON
SMOVL C01126 BC01126 V=11.7  +MOVJ EC01126
ARCOF
SMOVL C01127 BC01127 V=800.0  +MOVJ EC01127
SMOVL C01128 BC01128 V=1000.0  +MOVJ EC01128
SFTOF3D
'EndPath W4163
MOVJ C01129 BC01129 VJ=100.00  +MOVJ EC01129 VJ=100.00
'Path W4164
SFTOF3D
SFTON3D P041
MOVJ C01130 BC01130 VJ=100.00  +MOVJ EC01130 VJ=100.00
SMOVL C01131 BC01131 V=800.0  +MOVJ EC01131
SMOVL C01132 BC01132 V=150.0 PL=0  +MOVJ EC01132
MACRO1 MJ#(0) ARGF14
ARCON
SMOVL C01133 BC01133 V=10.0  +MOVJ EC01133
SMOVL C01134 BC01134 V=10.0  +MOVJ EC01134
SMOVL C01135 BC01135 V=10.0  +MOVJ EC01135
ARCOF
SMOVL C01136 BC01136 V=800.0  +MOVJ EC01136
SMOVL C01137 BC01137 V=1000.0  +MOVJ EC01137
SFTOF3D
'EndPath W4164
JUMP *L_1
'Path W4165
SFTOF3D
SFTON3D P041
MOVJ C01138 BC01138 VJ=100.00  +MOVJ EC01138 VJ=100.00
SMOVL C01139 BC01139 V=800.0  +MOVJ EC01139
SMOVL C01140 BC01140 V=150.0 PL=0  +MOVJ EC01140
SMOVL C01141 BC01141 V=10.0  +MOVJ EC01141
ARCOF
SMOVL C01142 BC01142 V=800.0  +MOVJ EC01142
SMOVL C01143 BC01143 V=1000.0  +MOVJ EC01143
SFTOF3D
'EndPath W4165
MOVJ C01144 BC01144 VJ=100.00  +MOVJ EC01144 VJ=100.00
'Path W4166
SFTOF3D
SFTON3D P041
MOVJ C01145 BC01145 VJ=100.00  +MOVJ EC01145 VJ=100.00
SMOVL C01146 BC01146 V=800.0  +MOVJ EC01146
SMOVL C01147 BC01147 V=150.0 PL=0  +MOVJ EC01147
SMOVL C01148 BC01148 V=10.0  +MOVJ EC01148
ARCOF
SMOVL C01149 BC01149 V=800.0  +MOVJ EC01149
SMOVL C01150 BC01150 V=1000.0  +MOVJ EC01150
SFTOF3D
'EndPath W4166
*L_1
MOVJ C01151 BC01151 VJ=100.00  +MOVJ EC01151 VJ=100.00
MOVJ C01152 BC01152 VJ=100.00  +MOVJ EC01152 VJ=100.00
MOVJ C01153 BC01153 VJ=100.00  +MOVJ EC01153 VJ=100.00
END
